LIN {X 0,Y 531.84,Z 443.101,A -85,B 0,C 180,E1 -4218.016,E2 -4218.016} C_VEL
LIN {X 0,Y 531.604,Z 454.409,A -85,B 0,C 180,E1 -4218.756,E2 -4218.756} C_VEL
LIN {X 0,Y 531.318,Z 464.837,A -85,B 0,C 180,E1 -4219.618,E2 -4219.618} C_VEL
LIN {X 0,Y 531.073,Z 475.093,A -85,B 0,C 180,E1 -4220.671,E2 -4220.671} C_VEL
LIN {X 0,Y 530.873,Z 483.99,A -85,B 0,C 180,E1 -4221.819,E2 -4221.819} C_VEL
LIN {X 0,Y 530.696,Z 491.14,A -85,B 0,C 180,E1 -4222.965,E2 -4222.965} C_VEL
LIN {X 0,Y 530.656,Z 495.995,A -85,B 0,C 180,E1 -4223.919,E2 -4223.919} C_VEL
LIN {X 0,Y 530.466,Z 500.698,A -85,B 0,C 180,E1 -4225.061,E2 -4225.061} C_VEL
LIN {X 0,Y 530.516,Z 504.289,A -85,B 0,C 180,E1 -4226.203,E2 -4226.203} C_VEL
LIN {X 0,Y 530.512,Z 506.139,A -85,B 0,C 180,E1 -4226.963,E2 -4226.963} C_VEL
LIN {X 0,Y 530.412,Z 507.563,A -85,B 0,C 180,E1 -4227.723,E2 -4227.723} C_VEL
LIN {X 0,Y 530.351,Z 509.173,A -85,B 0,C 180,E1 -4229.241,E2 -4229.241} C_VEL
LIN {X 0,Y 530.351,Z 509.411,A -85,B 0,C 180,E1 -4230.001,E2 -4230.001} C_VEL
LIN {X 0,Y 530.35,Z 509.227,A -85,B 0,C 180,E1 -4230.76,E2 -4230.76} C_VEL
LIN {X 0,Y 530.413,Z 507.691,A -85,B 0,C 180,E1 -4232.279,E2 -4232.279} C_VEL
LIN {X 0,Y 530.513,Z 506.338,A -85,B 0,C 180,E1 -4233.038,E2 -4233.038} C_VEL
LIN {X 0,Y 530.524,Z 503.495,A -85,B 0,C 180,E1 -4234.179,E2 -4234.179} C_VEL
LIN {X 0,Y 530.524,Z 499.631,A -85,B 0,C 180,E1 -4235.321,E2 -4235.321} C_VEL
LIN {X 0,Y 530.634,Z 493.865,A -85,B 0,C 180,E1 -4236.614,E2 -4236.614} C_VEL
LIN {X 0,Y 530.793,Z 487.123,A -85,B 0,C 180,E1 -4237.801,E2 -4237.801} C_VEL
LIN {X 0,Y 530.99,Z 478.999,A -85,B 0,C 180,E1 -4238.948,E2 -4238.948} C_VEL
LIN {X 0,Y 531.181,Z 470.63,A -85,B 0,C 180,E1 -4239.905,E2 -4239.905} C_VEL
LIN {X 0,Y 531.448,Z 460.37,A -85,B 0,C 180,E1 -4240.863,E2 -4240.863} C_VEL
LIN {X 0,Y 531.706,Z 449.647,A -85,B 0,C 180,E1 -4241.669,E2 -4241.669} C_VEL
LIN {X 0,Y 531.929,Z 439.01,A -85,B 0,C 180,E1 -4242.302,E2 -4242.302} C_VEL
LIN {X 0,Y 532.142,Z 426.406,A -85,B 0,C 180,E1 -4242.878,E2 -4242.878} C_VEL
LIN {X 0,Y 532.35,Z 413.949,A -85,B 0,C 180,E1 -4243.286,E2 -4243.286} C_VEL
LIN {X 0,Y 532.493,Z 401.048,A -85,B 0,C 180,E1 -4243.549,E2 -4243.549} C_VEL
LIN {X 0,Y 532.729,Z 307.619,A -85,B 0,C 180,E1 -4244.818,E2 -4244.818} C_VEL
LIN {X 0,Y 530.943,Z 296.994,A -85,B 0,C 180,E1 -4245.036,E2 -4245.036} C_VEL
LIN {X 0,Y 530.99,Z 279.347,A -85,B 0,C 180,E1 -4247.614,E2 -4247.614} C_VEL
LIN {X 0,Y 531.03,Z 279.335,A -85,B 0,C 180,E1 -4250.128,E2 -4250.128} C_VEL
LIN {X 0,Y 530.951,Z 279.344,A -85,B 0,C 180,E1 -4252.574,E2 -4252.574} C_VEL
LIN {X 0,Y 530.994,Z 279.343,A -85,B 0,C 180,E1 -4255.059,E2 -4255.059} C_VEL
LIN {X 0,Y 531.014,Z 279.341,A -85,B 0,C 180,E1 -4257.596,E2 -4257.596} C_VEL
LIN {X 0,Y 530.971,Z 279.342,A -85,B 0,C 180,E1 -4260.644,E2 -4260.644} C_VEL
LIN {X 0,Y 530.967,Z 279.347,A -85,B 0,C 180,E1 -4263.5,E2 -4263.5} C_VEL
LIN {X 0,Y 530.96,Z 279.344,A -85,B 0,C 180,E1 -4266.559,E2 -4266.559} C_VEL
LIN {X 0,Y 530.99,Z 279.343,A -85,B 0,C 180,E1 -4269.444,E2 -4269.444} C_VEL
LIN {X 0,Y 530.983,Z 279.341,A -85,B 0,C 180,E1 -4272.457,E2 -4272.457} C_VEL
LIN {X 0,Y 530.988,Z 279.34,A -85,B 0,C 180,E1 -4275.622,E2 -4275.622} C_VEL
LIN {X 0,Y 530.998,Z 279.341,A -85,B 0,C 180,E1 -4278.565,E2 -4278.565} C_VEL
LIN {X 0,Y 530.963,Z 279.343,A -85,B 0,C 180,E1 -4281.53,E2 -4281.53} C_VEL
LIN {X 0,Y 530.959,Z 279.344,A -85,B 0,C 180,E1 -4284.38,E2 -4284.38} C_VEL
LIN {X 0,Y 530.972,Z 279.345,A -85,B 0,C 180,E1 -4287.134,E2 -4287.134} C_VEL
LIN {X 0,Y 530.973,Z 279.34,A -85,B 0,C 180,E1 -4289.803,E2 -4289.803} C_VEL
LIN {X 0,Y 531.013,Z 279.34,A -85,B 0,C 180,E1 -4292.469,E2 -4292.469} C_VEL
LIN {X 0,Y 530.994,Z 279.343,A -85,B 0,C 180,E1 -4294.942,E2 -4294.942} C_VEL
LIN {X 0,Y 530.976,Z 279.343,A -85,B 0,C 180,E1 -4298.247,E2 -4298.247} C_VEL
LIN {X 0,Y 531.029,Z 279.405,A -85,B 0,C 180,E1 -4301.03,E2 -4301.03} C_VEL
LIN {X 0,Y 531.428,Z 285.13,A -85,B 0,C 180,E1 -4302.211,E2 -4302.211} C_VEL
LIN {X 0,Y 531.168,Z 299.568,A -85,B 0,C 180,E1 -4305.116,E2 -4305.116} C_VEL
LIN {X 0,Y 532.806,Z 309.363,A -85,B 0,C 180,E1 -4305.312,E2 -4305.312} C_VEL
LIN {X 0,Y 532.304,Z 405.637,A -85,B 0,C 180,E1 -4306.665,E2 -4306.665} C_VEL
LIN {X 0,Y 532.214,Z 419.063,A -85,B 0,C 180,E1 -4307.003,E2 -4307.003} C_VEL
LIN {X 0,Y 531.973,Z 431.141,A -85,B 0,C 180,E1 -4307.458,E2 -4307.458} C_VEL
LIN {X 0,Y 531.773,Z 443.346,A -85,B 0,C 180,E1 -4308.079,E2 -4308.079} C_VEL
LIN {X 0,Y 531.504,Z 456.293,A -85,B 0,C 180,E1 -4308.946,E2 -4308.946} C_VEL
LIN {X 0,Y 531.274,Z 465.371,A -85,B 0,C 180,E1 -4309.713,E2 -4309.713} C_VEL
LIN {X 0,Y 531.065,Z 474.673,A -85,B 0,C 180,E1 -4310.67,E2 -4310.67} C_VEL
LIN {X 0,Y 530.876,Z 482.343,A -85,B 0,C 180,E1 -4311.627,E2 -4311.627} C_VEL
LIN {X 0,Y 530.723,Z 489.883,A -85,B 0,C 180,E1 -4312.773,E2 -4312.773} C_VEL
LIN {X 0,Y 530.644,Z 495.898,A -85,B 0,C 180,E1 -4313.918,E2 -4313.918} C_VEL
LIN {X 0,Y 530.473,Z 500.651,A -85,B 0,C 180,E1 -4315.06,E2 -4315.06} C_VEL
LIN {X 0,Y 530.517,Z 504.276,A -85,B 0,C 180,E1 -4316.202,E2 -4316.202} C_VEL
LIN {X 0,Y 530.512,Z 506.099,A -85,B 0,C 180,E1 -4316.962,E2 -4316.962} C_VEL
LIN {X 0,Y 530.362,Z 508.579,A -85,B 0,C 180,E1 -4318.481,E2 -4318.481} C_VEL
LIN {X 0,Y 530.352,Z 509.18,A -85,B 0,C 180,E1 -4319.241,E2 -4319.241} C_VEL
LIN {X 0,Y 530.352,Z 509.246,A -85,B 0,C 180,E1 -4320.759,E2 -4320.759} C_VEL
LIN {X 0,Y 530.362,Z 508.673,A -85,B 0,C 180,E1 -4321.519,E2 -4321.519} C_VEL
LIN {X 0,Y 530.513,Z 506.338,A -85,B 0,C 180,E1 -4323.038,E2 -4323.038} C_VEL
LIN {X 0,Y 530.524,Z 503.472,A -85,B 0,C 180,E1 -4324.178,E2 -4324.178} C_VEL
LIN {X 0,Y 530.524,Z 499.567,A -85,B 0,C 180,E1 -4325.321,E2 -4325.321} C_VEL
LIN {X 0,Y 530.618,Z 495.221,A -85,B 0,C 180,E1 -4326.325,E2 -4326.325} C_VEL
LIN {X 0,Y 530.73,Z 489.328,A -85,B 0,C 180,E1 -4327.418,E2 -4327.418} C_VEL
LIN {X 0,Y 530.853,Z 483.075,A -85,B 0,C 180,E1 -4328.374,E2 -4328.374} C_VEL
LIN {X 0,Y 531.05,Z 475.529,A -85,B 0,C 180,E1 -4329.33,E2 -4329.33} C_VEL
LIN {X 0,Y 531.24,Z 466.368,A -85,B 0,C 180,E1 -4330.288,E2 -4330.288} C_VEL
LIN {X 0,Y 531.521,Z 456.247,A -85,B 0,C 180,E1 -4331.15,E2 -4331.15} C_VEL
LIN {X 0,Y 531.755,Z 444.083,A -85,B 0,C 180,E1 -4331.968,E2 -4331.968} C_VEL
LIN {X 0,Y 531.941,Z 431.979,A -85,B 0,C 180,E1 -4332.591,E2 -4332.591} C_VEL
LIN {X 0,Y 532.15,Z 418.568,A -85,B 0,C 180,E1 -4333.096,E2 -4333.096} C_VEL
LIN {X 0,Y 532.315,Z 406.003,A -85,B 0,C 180,E1 -4333.407,E2 -4333.407} C_VEL
LIN {X 0,Y 532.63,Z 307.356,A -85,B 0,C 180,E1 -4334.813,E2 -4334.813} C_VEL
LIN {X 0,Y 531.242,Z 300.133,A -85,B 0,C 180,E1 -4334.97,E2 -4334.97} C_VEL
LIN {X 0,Y 531.56,Z 285.055,A -85,B 0,C 180,E1 -4338.062,E2 -4338.062} C_VEL
LIN {X 0,Y 531.04,Z 279.34,A -85,B 0,C 180,E1 -4339.321,E2 -4339.321} C_VEL
LIN {X 0,Y 530.98,Z 279.343,A -85,B 0,C 180,E1 -4342.101,E2 -4342.101} C_VEL
LIN {X 0,Y 530.942,Z 279.352,A -85,B 0,C 180,E1 -4345.061,E2 -4345.061} C_VEL
LIN {X 0,Y 530.953,Z 279.348,A -85,B 0,C 180,E1 -4347.599,E2 -4347.599} C_VEL
LIN {X 0,Y 530.944,Z 279.349,A -85,B 0,C 180,E1 -4350.639,E2 -4350.639} C_VEL
LIN {X 0,Y 530.948,Z 279.347,A -85,B 0,C 180,E1 -4353.496,E2 -4353.496} C_VEL
LIN {X 0,Y 530.9,Z 279.351,A -85,B 0,C 180,E1 -4356.146,E2 -4356.146} C_VEL
LIN {X 0,Y 530.954,Z 279.344,A -85,B 0,C 180,E1 -4359.446,E2 -4359.446} C_VEL
LIN {X 0,Y 530.916,Z 279.354,A -85,B 0,C 180,E1 -4362.463,E2 -4362.463} C_VEL
LIN {X 0,Y 530.963,Z 279.342,A -85,B 0,C 180,E1 -4365.45,E2 -4365.45} C_VEL
LIN {X 0,Y 530.953,Z 279.35,A -85,B 0,C 180,E1 -4368.56,E2 -4368.56} C_VEL
LIN {X 0,Y 530.953,Z 279.344,A -85,B 0,C 180,E1 -4371.528,E2 -4371.528} C_VEL
LIN {X 0,Y 530.951,Z 279.351,A -85,B 0,C 180,E1 -4374.379,E2 -4374.379} C_VEL
LIN {X 0,Y 530.971,Z 279.343,A -85,B 0,C 180,E1 -4377.133,E2 -4377.133} C_VEL
LIN {X 0,Y 530.958,Z 279.352,A -85,B 0,C 180,E1 -4379.802,E2 -4379.802} C_VEL
LIN {X 0,Y 530.971,Z 279.346,A -85,B 0,C 180,E1 -4382.477,E2 -4382.477} C_VEL
LIN {X 0,Y 531.061,Z 279.462,A -85,B 0,C 180,E1 -4385.232,E2 -4385.232} C_VEL
LIN {X 0,Y 532.337,Z 287.063,A -85,B 0,C 180,E1 -4386.461,E2 -4386.461} C_VEL
LIN {X 0,Y 532.028,Z 303.307,A -85,B 0,C 180,E1 -4388.901,E2 -4388.901} C_VEL
LIN {X 0,Y 531.681,Z 322.238,A -85,B 0,C 180,E1 -4391.695,E2 -4391.695} C_VEL
LIN {X 0,Y 531.362,Z 341.292,A -85,B 0,C 180,E1 -4394.464,E2 -4394.464} C_VEL
LIN {X 0,Y 531.274,Z 345.358,A -85,B 0,C 180,E1 -4395.052,E2 -4395.052} C_VEL
LIN {X 0,Y 532.724,Z 356.776,A -85,B 0,C 180,E1 -4395.271,E2 -4395.271} C_VEL
LIN {X 0,Y 532.333,Z 452.199,A -85,B 0,C 180,E1 -4396.592,E2 -4396.592} C_VEL
LIN {X 0,Y 532.128,Z 464.759,A -85,B 0,C 180,E1 -4396.879,E2 -4396.879} C_VEL
LIN {X 0,Y 531.919,Z 478.246,A -85,B 0,C 180,E1 -4397.359,E2 -4397.359} C_VEL
LIN {X 0,Y 531.758,Z 489.353,A -85,B 0,C 180,E1 -4397.896,E2 -4397.896} C_VEL
LIN {X 0,Y 531.519,Z 500.184,A -85,B 0,C 180,E1 -4398.56,E2 -4398.56} C_VEL
LIN {X 0,Y 531.267,Z 511.362,A -85,B 0,C 180,E1 -4399.423,E2 -4399.423} C_VEL
LIN {X 0,Y 531.049,Z 520.423,A -85,B 0,C 180,E1 -4400.285,E2 -4400.285} C_VEL
LIN {X 0,Y 530.835,Z 530.246,A -85,B 0,C 180,E1 -4401.434,E2 -4401.434} C_VEL
LIN {X 0,Y 530.675,Z 538.064,A -85,B 0,C 180,E1 -4402.58,E2 -4402.58} C_VEL
LIN {X 0,Y 530.585,Z 545.242,A -85,B 0,C 180,E1 -4403.916,E2 -4403.916} C_VEL
LIN {X 0,Y 530.459,Z 550.013,A -85,B 0,C 180,E1 -4405.059,E2 -4405.059} C_VEL
LIN {X 0,Y 530.516,Z 553.668,A -85,B 0,C 180,E1 -4406.201,E2 -4406.201} C_VEL
LIN {X 0,Y 530.457,Z 555.549,A -85,B 0,C 180,E1 -4406.961,E2 -4406.961} C_VEL
LIN {X 0,Y 530.411,Z 556.955,A -85,B 0,C 180,E1 -4407.721,E2 -4407.721} C_VEL
LIN {X 0,Y 530.345,Z 558.568,A -85,B 0,C 180,E1 -4409.24,E2 -4409.24} C_VEL
LIN {X 0,Y 530.346,Z 558.788,A -85,B 0,C 180,E1 -4409.999,E2 -4409.999} C_VEL
LIN {X 0,Y 530.361,Z 557.962,A -85,B 0,C 180,E1 -4411.518,E2 -4411.518} C_VEL
LIN {X 0,Y 530.411,Z 556.964,A -85,B 0,C 180,E1 -4412.277,E2 -4412.277} C_VEL
LIN {X 0,Y 530.457,Z 555.561,A -85,B 0,C 180,E1 -4413.037,E2 -4413.037} C_VEL
LIN {X 0,Y 530.522,Z 552.614,A -85,B 0,C 180,E1 -4414.177,E2 -4414.177} C_VEL
LIN {X 0,Y 530.524,Z 548.615,A -85,B 0,C 180,E1 -4415.32,E2 -4415.32} C_VEL
LIN {X 0,Y 530.598,Z 542.845,A -85,B 0,C 180,E1 -4416.581,E2 -4416.581} C_VEL
LIN {X 0,Y 530.719,Z 535.717,A -85,B 0,C 180,E1 -4417.8,E2 -4417.8} C_VEL
LIN {X 0,Y 530.912,Z 527.353,A -85,B 0,C 180,E1 -4418.947,E2 -4418.947} C_VEL
LIN {X 0,Y 531.081,Z 518.752,A -85,B 0,C 180,E1 -4419.905,E2 -4419.905} C_VEL
LIN {X 0,Y 531.356,Z 508.129,A -85,B 0,C 180,E1 -4420.863,E2 -4420.863} C_VEL
LIN {X 0,Y 531.567,Z 497.005,A -85,B 0,C 180,E1 -4421.671,E2 -4421.671} C_VEL
LIN {X 0,Y 531.822,Z 486.007,A -85,B 0,C 180,E1 -4422.303,E2 -4422.303} C_VEL
LIN {X 0,Y 532.037,Z 473.98,A -85,B 0,C 180,E1 -4422.831,E2 -4422.831} C_VEL
LIN {X 0,Y 532.209,Z 460.97,A -85,B 0,C 180,E1 -4423.239,E2 -4423.239} C_VEL
LIN {X 0,Y 532.392,Z 447.236,A -85,B 0,C 180,E1 -4423.502,E2 -4423.502} C_VEL
LIN {X 0,Y 532.666,Z 354.778,A -85,B 0,C 180,E1 -4424.767,E2 -4424.767} C_VEL
LIN {X 0,Y 531.319,Z 345.814,A -85,B 0,C 180,E1 -4424.952,E2 -4424.952} C_VEL
LIN {X 0,Y 531.679,Z 327.116,A -85,B 0,C 180,E1 -4427.699,E2 -4427.699} C_VEL
LIN {X 0,Y 532.152,Z 305.555,A -85,B 0,C 180,E1 -4430.889,E2 -4430.889} C_VEL
LIN {X 0,Y 532.585,Z 288.083,A -85,B 0,C 180,E1 -4433.526,E2 -4433.526} C_VEL
LIN {X 0,Y 531.04,Z 279.338,A -85,B 0,C 180,E1 -4434.976,E2 -4434.976} C_VEL
LIN {X 0,Y 531.007,Z 279.341,A -85,B 0,C 180,E1 -4437.595,E2 -4437.595} C_VEL
LIN {X 0,Y 530.972,Z 279.341,A -85,B 0,C 180,E1 -4440.644,E2 -4440.644} C_VEL
LIN {X 0,Y 530.984,Z 279.345,A -85,B 0,C 180,E1 -4443.772,E2 -4443.772} C_VEL
LIN {X 0,Y 530.946,Z 279.344,A -85,B 0,C 180,E1 -4446.558,E2 -4446.558} C_VEL
LIN {X 0,Y 530.981,Z 279.343,A -85,B 0,C 180,E1 -4449.443,E2 -4449.443} C_VEL
LIN {X 0,Y 530.958,Z 279.343,A -85,B 0,C 180,E1 -4452.457,E2 -4452.457} C_VEL
LIN {X 0,Y 530.962,Z 279.347,A -85,B 0,C 180,E1 -4455.45,E2 -4455.45} C_VEL
LIN {X 0,Y 530.974,Z 279.34,A -85,B 0,C 180,E1 -4458.562,E2 -4458.562} C_VEL
LIN {X 0,Y 530.947,Z 279.352,A -85,B 0,C 180,E1 -4461.528,E2 -4461.528} C_VEL
LIN {X 0,Y 530.946,Z 279.344,A -85,B 0,C 180,E1 -4464.379,E2 -4464.379} C_VEL
LIN {X 0,Y 530.958,Z 279.348,A -85,B 0,C 180,E1 -4467.133,E2 -4467.133} C_VEL
LIN {X 0,Y 530.942,Z 279.347,A -85,B 0,C 180,E1 -4469.801,E2 -4469.801} C_VEL
LIN {X 0,Y 530.955,Z 279.344,A -85,B 0,C 180,E1 -4472.477,E2 -4472.477} C_VEL
LIN {X 0,Y 530.938,Z 279.35,A -85,B 0,C 180,E1 -4474.939,E2 -4474.939} C_VEL
LIN {X 0,Y 530.967,Z 279.342,A -85,B 0,C 180,E1 -4477.898,E2 -4477.898} C_VEL
LIN {X 0,Y 530.972,Z 279.345,A -85,B 0,C 180,E1 -4480.676,E2 -4480.676} C_VEL
LIN {X 0,Y 530.949,Z 279.351,A -85,B 0,C 180,E1 -4483.07,E2 -4483.07} C_VEL
LIN {X 0,Y 530.988,Z 279.341,A -85,B 0,C 180,E1 -4485.435,E2 -4485.435} C_VEL
LIN {X 0,Y 531.02,Z 279.34,A -85,B 0,C 180,E1 -4488.549,E2 -4488.549} C_VEL
LIN {X 0,Y 531.018,Z 279.336,A -85,B 0,C 180,E1 -4491.629,E2 -4491.629} C_VEL
LIN {X 0,Y 531.072,Z 279.335,A -85,B 0,C 180,E1 -4494.685,E2 -4494.685} C_VEL
LIN {X 0,Y 531.113,Z 279.324,A -85,B 0,C 180,E1 -4497.725,E2 -4497.725} C_VEL
LIN {X 0,Y 531.138,Z 279.325,A -85,B 0,C 180,E1 -4500.758,E2 -4500.758} C_VEL
LIN {X 0,Y 531.045,Z 279.334,A -85,B 0,C 180,E1 -4503.035,E2 -4503.035} C_VEL
LIN {X 0,Y 531.031,Z 279.339,A -85,B 0,C 180,E1 -4506.078,E2 -4506.078} C_VEL
LIN {X 0,Y 530.996,Z 279.339,A -85,B 0,C 180,E1 -4509.139,E2 -4509.139} C_VEL
LIN {X 0,Y 531.039,Z 279.336,A -85,B 0,C 180,E1 -4511.67,E2 -4511.67} C_VEL
LIN {X 0,Y 531.014,Z 279.337,A -85,B 0,C 180,E1 -4514.953,E2 -4514.953} C_VEL
LIN {X 0,Y 530.971,Z 279.347,A -85,B 0,C 180,E1 -4517.724,E2 -4517.724} C_VEL
LIN {X 0,Y 531.016,Z 279.342,A -85,B 0,C 180,E1 -4520.128,E2 -4520.128} C_VEL
LIN {X 0,Y 530.936,Z 279.347,A -85,B 0,C 180,E1 -4522.574,E2 -4522.574} C_VEL
LIN {X 0,Y 530.978,Z 279.342,A -85,B 0,C 180,E1 -4525.059,E2 -4525.059} C_VEL
LIN {X 0,Y 530.957,Z 279.349,A -85,B 0,C 180,E1 -4527.599,E2 -4527.599} C_VEL
LIN {X 0,Y 530.953,Z 279.346,A -85,B 0,C 180,E1 -4530.198,E2 -4530.198} C_VEL
LIN {X 0,Y 530.96,Z 279.344,A -85,B 0,C 180,E1 -4532.867,E2 -4532.867} C_VEL
LIN {X 0,Y 530.943,Z 279.351,A -85,B 0,C 180,E1 -4535.621,E2 -4535.621} C_VEL
LIN {X 0,Y 530.957,Z 279.344,A -85,B 0,C 180,E1 -4538.654,E2 -4538.654} C_VEL
LIN {X 0,Y 530.983,Z 279.346,A -85,B 0,C 180,E1 -4541.437,E2 -4541.437} C_VEL
LIN {X 0,Y 530.937,Z 279.35,A -85,B 0,C 180,E1 -4543.56,E2 -4543.56} C_VEL
LIN {X 0,Y 530.27,Z 279.43,A -85,B 0,C 180,E1 -4544.193,E2 -4544.193} C_VEL
LIN {X 0,Y 527.427,Z 279.789,A -85,B 0,C 180,E1 -4545.222,E2 -4545.222} C_VEL
LIN {X 0,Y 525.026,Z 280.088,A -85,B 0,C 180,E1 -4546.051,E2 -4546.051} C_VEL
LIN {X 0,Y 523.995,Z 280.215,A -85,B 0,C 180,E1 -4546.691,E2 -4546.691} C_VEL
LIN {X 0,Y 523.91,Z 280.225,A -85,B 0,C 180,E1 -4546.907,E2 -4546.907} C_VEL
LIN {X 0,Y 523.945,Z 280.218,A -85,B 0,C 180,E1 -4549.922,E2 -4549.922} C_VEL
LIN {X 0,Y 523.904,Z 280.228,A -85,B 0,C 180,E1 -4552.869,E2 -4552.869} C_VEL
LIN {X 0,Y 523.917,Z 280.222,A -85,B 0,C 180,E1 -4555.71,E2 -4555.71} C_VEL
LIN {X 0,Y 523.917,Z 280.223,A -85,B 0,C 180,E1 -4558.457,E2 -4558.457} C_VEL
LIN {X 0,Y 523.928,Z 280.224,A -85,B 0,C 180,E1 -4561.126,E2 -4561.126} C_VEL
LIN {X 0,Y 523.983,Z 280.213,A -85,B 0,C 180,E1 -4563.981,E2 -4563.981} C_VEL
LIN {X 0,Y 523.911,Z 280.225,A -85,B 0,C 180,E1 -4567.107,E2 -4567.107} C_VEL
LIN {X 0,Y 523.979,Z 280.213,A -85,B 0,C 180,E1 -4569.867,E2 -4569.867} C_VEL
LIN {X 0,Y 523.902,Z 280.231,A -85,B 0,C 180,E1 -4572.601,E2 -4572.601} C_VEL
LIN {X 0,Y 523.873,Z 295.889,A -85,B 0,C 180,E1 -4574.771,E2 -4574.771} C_VEL
LIN {X 0,Y 523.904,Z 296.55,A -85,B 0,C 180,E1 -4574.856,E2 -4574.856} C_VEL
LIN {X 0,Y 525.989,Z 309.337,A -85,B 0,C 180,E1 -4575.099,E2 -4575.099} C_VEL
LIN {X 0,Y 525.543,Z 405.952,A -85,B 0,C 180,E1 -4576.442,E2 -4576.442} C_VEL
LIN {X 0,Y 525.379,Z 419.475,A -85,B 0,C 180,E1 -4576.782,E2 -4576.782} C_VEL
LIN {X 0,Y 525.135,Z 431.546,A -85,B 0,C 180,E1 -4577.243,E2 -4577.243} C_VEL
LIN {X 0,Y 524.898,Z 444.027,A -85,B 0,C 180,E1 -4577.892,E2 -4577.892} C_VEL
LIN {X 0,Y 524.661,Z 454.714,A -85,B 0,C 180,E1 -4578.605,E2 -4578.605} C_VEL
LIN {X 0,Y 524.33,Z 465.146,A -85,B 0,C 180,E1 -4579.478,E2 -4579.478} C_VEL
LIN {X 0,Y 524.078,Z 475.405,A -85,B 0,C 180,E1 -4580.546,E2 -4580.546} C_VEL
LIN {X 0,Y 523.84,Z 484.305,A -85,B 0,C 180,E1 -4581.708,E2 -4581.708} C_VEL
LIN {X 0,Y 523.659,Z 491.456,A -85,B 0,C 180,E1 -4582.87,E2 -4582.87} C_VEL
LIN {X 0,Y 523.601,Z 496.312,A -85,B 0,C 180,E1 -4583.837,E2 -4583.837} C_VEL
LIN {X 0,Y 523.392,Z 501.016,A -85,B 0,C 180,E1 -4584.994,E2 -4584.994} C_VEL
LIN {X 0,Y 523.443,Z 504.606,A -85,B 0,C 180,E1 -4586.152,E2 -4586.152} C_VEL
LIN {X 0,Y 523.446,Z 506.456,A -85,B 0,C 180,E1 -4586.922,E2 -4586.922} C_VEL
LIN {X 0,Y 523.338,Z 507.88,A -85,B 0,C 180,E1 -4587.692,E2 -4587.692} C_VEL
LIN {X 0,Y 523.259,Z 509.49,A -85,B 0,C 180,E1 -4589.231,E2 -4589.231} C_VEL
LIN {X 0,Y 523.259,Z 509.728,A -85,B 0,C 180,E1 -4590.001,E2 -4590.001} C_VEL
LIN {X 0,Y 523.258,Z 509.544,A -85,B 0,C 180,E1 -4590.77,E2 -4590.77} C_VEL
LIN {X 0,Y 523.338,Z 508.006,A -85,B 0,C 180,E1 -4592.31,E2 -4592.31} C_VEL
LIN {X 0,Y 523.447,Z 506.652,A -85,B 0,C 180,E1 -4593.079,E2 -4593.079} C_VEL
LIN {X 0,Y 523.449,Z 503.809,A -85,B 0,C 180,E1 -4594.236,E2 -4594.236} C_VEL
LIN {X 0,Y 523.464,Z 499.943,A -85,B 0,C 180,E1 -4595.393,E2 -4595.393} C_VEL
LIN {X 0,Y 523.564,Z 494.602,A -85,B 0,C 180,E1 -4596.619,E2 -4596.619} C_VEL
LIN {X 0,Y 523.773,Z 487.431,A -85,B 0,C 180,E1 -4597.906,E2 -4597.906} C_VEL
LIN {X 0,Y 523.965,Z 479.304,A -85,B 0,C 180,E1 -4599.069,E2 -4599.069} C_VEL
LIN {X 0,Y 524.188,Z 470.929,A -85,B 0,C 180,E1 -4600.038,E2 -4600.038} C_VEL
LIN {X 0,Y 524.483,Z 460.663,A -85,B 0,C 180,E1 -4601.009,E2 -4601.009} C_VEL
LIN {X 0,Y 524.751,Z 450.206,A -85,B 0,C 180,E1 -4601.807,E2 -4601.807} C_VEL
LIN {X 0,Y 525.008,Z 439.281,A -85,B 0,C 180,E1 -4602.466,E2 -4602.466} C_VEL
LIN {X 0,Y 525.243,Z 426.658,A -85,B 0,C 180,E1 -4603.05,E2 -4603.05} C_VEL
LIN {X 0,Y 525.47,Z 414.157,A -85,B 0,C 180,E1 -4603.463,E2 -4603.463} C_VEL
LIN {X 0,Y 525.606,Z 401.164,A -85,B 0,C 180,E1 -4603.73,E2 -4603.73} C_VEL
LIN {X 0,Y 525.987,Z 309.161,A -85,B 0,C 180,E1 -4604.993,E2 -4604.993} C_VEL
LIN {X 0,Y 523.876,Z 296.59,A -85,B 0,C 180,E1 -4605.233,E2 -4605.233} C_VEL
LIN {X 0,Y 523.869,Z 281.402,A -85,B 0,C 180,E1 -4607.318,E2 -4607.318} C_VEL
LIN {X 0,Y 523.867,Z 280.235,A -85,B 0,C 180,E1 -4607.514,E2 -4607.514} C_VEL
LIN {X 0,Y 523.984,Z 280.213,A -85,B 0,C 180,E1 -4610.134,E2 -4610.134} C_VEL
LIN {X 0,Y 523.916,Z 280.223,A -85,B 0,C 180,E1 -4612.894,E2 -4612.894} C_VEL
LIN {X 0,Y 523.988,Z 280.212,A -85,B 0,C 180,E1 -4616.02,E2 -4616.02} C_VEL
LIN {X 0,Y 523.934,Z 280.221,A -85,B 0,C 180,E1 -4618.876,E2 -4618.876} C_VEL
LIN {X 0,Y 523.924,Z 280.224,A -85,B 0,C 180,E1 -4621.545,E2 -4621.545} C_VEL
LIN {X 0,Y 523.925,Z 280.219,A -85,B 0,C 180,E1 -4624.292,E2 -4624.292} C_VEL
LIN {X 0,Y 523.912,Z 280.227,A -85,B 0,C 180,E1 -4627.133,E2 -4627.133} C_VEL
LIN {X 0,Y 523.943,Z 280.217,A -85,B 0,C 180,E1 -4630.13,E2 -4630.13} C_VEL
LIN {X 0,Y 523.927,Z 280.226,A -85,B 0,C 180,E1 -4633.167,E2 -4633.167} C_VEL
LIN {X 0,Y 523.941,Z 280.217,A -85,B 0,C 180,E1 -4635.772,E2 -4635.772} C_VEL
LIN {X 0,Y 523.944,Z 280.223,A -85,B 0,C 180,E1 -4638.908,E2 -4638.908} C_VEL
LIN {X 0,Y 523.921,Z 280.219,A -85,B 0,C 180,E1 -4641.898,E2 -4641.898} C_VEL
LIN {X 0,Y 523.929,Z 280.226,A -85,B 0,C 180,E1 -4644.911,E2 -4644.911} C_VEL
LIN {X 0,Y 523.94,Z 280.216,A -85,B 0,C 180,E1 -4647.68,E2 -4647.68} C_VEL
LIN {X 0,Y 523.958,Z 280.221,A -85,B 0,C 180,E1 -4650.677,E2 -4650.677} C_VEL
LIN {X 0,Y 523.95,Z 280.222,A -85,B 0,C 180,E1 -4652.867,E2 -4652.867} C_VEL
LIN {X 0,Y 523.946,Z 280.215,A -85,B 0,C 180,E1 -4655.802,E2 -4655.802} C_VEL
LIN {X 0,Y 523.95,Z 280.223,A -85,B 0,C 180,E1 -4658.767,E2 -4658.767} C_VEL
LIN {X 0,Y 523.994,Z 280.322,A -85,B 0,C 180,E1 -4660.918,E2 -4660.918} C_VEL
LIN {X 0,Y 524.447,Z 285.856,A -85,B 0,C 180,E1 -4662.075,E2 -4662.075} C_VEL
LIN {X 0,Y 524.182,Z 299.819,A -85,B 0,C 180,E1 -4664.913,E2 -4664.913} C_VEL
LIN {X 0,Y 525.952,Z 309.464,A -85,B 0,C 180,E1 -4665.116,E2 -4665.116} C_VEL
LIN {X 0,Y 525.383,Z 406.411,A -85,B 0,C 180,E1 -4666.511,E2 -4666.511} C_VEL
LIN {X 0,Y 525.278,Z 420.296,A -85,B 0,C 180,E1 -4666.877,E2 -4666.877} C_VEL
LIN {X 0,Y 525.013,Z 432.131,A -85,B 0,C 180,E1 -4667.338,E2 -4667.338} C_VEL
LIN {X 0,Y 524.795,Z 444.278,A -85,B 0,C 180,E1 -4667.974,E2 -4667.974} C_VEL
LIN {X 0,Y 524.536,Z 456.361,A -85,B 0,C 180,E1 -4668.797,E2 -4668.797} C_VEL
LIN {X 0,Y 524.265,Z 465.51,A -85,B 0,C 180,E1 -4669.573,E2 -4669.573} C_VEL
LIN {X 0,Y 524.036,Z 474.853,A -85,B 0,C 180,E1 -4670.544,E2 -4670.544} C_VEL
LIN {X 0,Y 523.857,Z 482.554,A -85,B 0,C 180,E1 -4671.514,E2 -4671.514} C_VEL
LIN {X 0,Y 523.665,Z 490.107,A -85,B 0,C 180,E1 -4672.675,E2 -4672.675} C_VEL
LIN {X 0,Y 523.577,Z 496.146,A -85,B 0,C 180,E1 -4673.835,E2 -4673.835} C_VEL
LIN {X 0,Y 523.395,Z 500.92,A -85,B 0,C 180,E1 -4674.993,E2 -4674.993} C_VEL
LIN {X 0,Y 523.444,Z 504.566,A -85,B 0,C 180,E1 -4676.151,E2 -4676.151} C_VEL
LIN {X 0,Y 523.447,Z 506.412,A -85,B 0,C 180,E1 -4676.921,E2 -4676.921} C_VEL
LIN {X 0,Y 523.275,Z 508.897,A -85,B 0,C 180,E1 -4678.461,E2 -4678.461} C_VEL
LIN {X 0,Y 523.261,Z 509.51,A -85,B 0,C 180,E1 -4679.23,E2 -4679.23} C_VEL
LIN {X 0,Y 523.26,Z 509.579,A -85,B 0,C 180,E1 -4680.77,E2 -4680.77} C_VEL
LIN {X 0,Y 523.275,Z 509.011,A -85,B 0,C 180,E1 -4681.539,E2 -4681.539} C_VEL
LIN {X 0,Y 523.447,Z 506.667,A -85,B 0,C 180,E1 -4683.079,E2 -4683.079} C_VEL
LIN {X 0,Y 523.449,Z 503.793,A -85,B 0,C 180,E1 -4684.235,E2 -4684.235} C_VEL
LIN {X 0,Y 523.463,Z 499.875,A -85,B 0,C 180,E1 -4685.393,E2 -4685.393} C_VEL
LIN {X 0,Y 523.561,Z 494.486,A -85,B 0,C 180,E1 -4686.615,E2 -4686.615} C_VEL
LIN {X 0,Y 523.705,Z 488.418,A -85,B 0,C 180,E1 -4687.712,E2 -4687.712} C_VEL
LIN {X 0,Y 523.924,Z 480.451,A -85,B 0,C 180,E1 -4688.874,E2 -4688.874} C_VEL
LIN {X 0,Y 524.13,Z 472.277,A -85,B 0,C 180,E1 -4689.844,E2 -4689.844} C_VEL
LIN {X 0,Y 524.369,Z 462.263,A -85,B 0,C 180,E1 -4690.815,E2 -4690.815} C_VEL
LIN {X 0,Y 524.666,Z 450.855,A -85,B 0,C 180,E1 -4691.692,E2 -4691.692} C_VEL
LIN {X 0,Y 524.896,Z 439.732,A -85,B 0,C 180,E1 -4692.37,E2 -4692.37} C_VEL
LIN {X 0,Y 525.098,Z 428.425,A -85,B 0,C 180,E1 -4692.906,E2 -4692.906} C_VEL
LIN {X 0,Y 525.291,Z 415.626,A -85,B 0,C 180,E1 -4693.344,E2 -4693.344} C_VEL
LIN {X 0,Y 525.4,Z 402.166,A -85,B 0,C 180,E1 -4693.636,E2 -4693.636} C_VEL
LIN {X 0,Y 525.898,Z 308.914,A -85,B 0,C 180,E1 -4694.982,E2 -4694.982} C_VEL
LIN {X 0,Y 524.283,Z 300.578,A -85,B 0,C 180,E1 -4695.168,E2 -4695.168} C_VEL
LIN {X 0,Y 524.6,Z 287.041,A -85,B 0,C 180,E1 -4697.976,E2 -4697.976} C_VEL
LIN {X 0,Y 524.188,Z 281.462,A -85,B 0,C 180,E1 -4699.177,E2 -4699.177} C_VEL
LIN {X 0,Y 523.984,Z 280.219,A -85,B 0,C 180,E1 -4699.49,E2 -4699.49} C_VEL
LIN {X 0,Y 523.92,Z 280.223,A -85,B 0,C 180,E1 -4702.242,E2 -4702.242} C_VEL
LIN {X 0,Y 523.9,Z 280.225,A -85,B 0,C 180,E1 -4704.573,E2 -4704.573} C_VEL
LIN {X 0,Y 523.914,Z 280.224,A -85,B 0,C 180,E1 -4707.704,E2 -4707.704} C_VEL
LIN {X 0,Y 523.9,Z 280.228,A -85,B 0,C 180,E1 -4710.845,E2 -4710.845} C_VEL
LIN {X 0,Y 523.912,Z 280.222,A -85,B 0,C 180,E1 -4713.726,E2 -4713.726} C_VEL
LIN {X 0,Y 523.858,Z 280.23,A -85,B 0,C 180,E1 -4716.394,E2 -4716.394} C_VEL
LIN {X 0,Y 523.9,Z 280.226,A -85,B 0,C 180,E1 -4719.087,E2 -4719.087} C_VEL
LIN {X 0,Y 523.894,Z 280.225,A -85,B 0,C 180,E1 -4722.125,E2 -4722.125} C_VEL
LIN {X 0,Y 523.934,Z 280.218,A -85,B 0,C 180,E1 -4725.311,E2 -4725.311} C_VEL
LIN {X 0,Y 523.915,Z 280.226,A -85,B 0,C 180,E1 -4728.695,E2 -4728.695} C_VEL
LIN {X 0,Y 523.914,Z 280.224,A -85,B 0,C 180,E1 -4731.897,E2 -4731.897} C_VEL
LIN {X 0,Y 523.922,Z 280.221,A -85,B 0,C 180,E1 -4734.912,E2 -4734.912} C_VEL
LIN {X 0,Y 523.939,Z 280.222,A -85,B 0,C 180,E1 -4737.679,E2 -4737.679} C_VEL
LIN {X 0,Y 523.956,Z 280.221,A -85,B 0,C 180,E1 -4740.677,E2 -4740.677} C_VEL
LIN {X 0,Y 523.935,Z 280.225,A -85,B 0,C 180,E1 -4743.726,E2 -4743.726} C_VEL
LIN {X 0,Y 523.997,Z 280.266,A -85,B 0,C 180,E1 -4745.034,E2 -4745.034} C_VEL
LIN {X 0,Y 525.376,Z 288.167,A -85,B 0,C 180,E1 -4746.339,E2 -4746.339} C_VEL
LIN {X 0,Y 525.196,Z 298.895,A -85,B 0,C 180,E1 -4747.994,E2 -4747.994} C_VEL
LIN {X 0,Y 524.772,Z 316.472,A -85,B 0,C 180,E1 -4750.642,E2 -4750.642} C_VEL
LIN {X 0,Y 524.448,Z 334.09,A -85,B 0,C 180,E1 -4753.254,E2 -4753.254} C_VEL
LIN {X 0,Y 524.268,Z 344.866,A -85,B 0,C 180,E1 -4754.838,E2 -4754.838} C_VEL
LIN {X 0,Y 525.862,Z 356.746,A -85,B 0,C 180,E1 -4755.08,E2 -4755.08} C_VEL
LIN {X 0,Y 525.385,Z 453.304,A -85,B 0,C 180,E1 -4756.461,E2 -4756.461} C_VEL
LIN {X 0,Y 525.165,Z 465.949,A -85,B 0,C 180,E1 -4756.775,E2 -4756.775} C_VEL
LIN {X 0,Y 524.891,Z 479.58,A -85,B 0,C 180,E1 -4757.285,E2 -4757.285} C_VEL
LIN {X 0,Y 524.68,Z 491.736,A -85,B 0,C 180,E1 -4757.912,E2 -4757.912} C_VEL
LIN {X 0,Y 524.372,Z 503.491,A -85,B 0,C 180,E1 -4758.695,E2 -4758.695} C_VEL
LIN {X 0,Y 524.153,Z 513.999,A -85,B 0,C 180,E1 -4759.571,E2 -4759.571} C_VEL
LIN {X 0,Y 523.905,Z 523.41,A -85,B 0,C 180,E1 -4760.541,E2 -4760.541} C_VEL
LIN {X 0,Y 523.704,Z 532.525,A -85,B 0,C 180,E1 -4761.705,E2 -4761.705} C_VEL
LIN {X 0,Y 523.573,Z 539.877,A -85,B 0,C 180,E1 -4762.867,E2 -4762.867} C_VEL
LIN {X 0,Y 523.48,Z 544.816,A -85,B 0,C 180,E1 -4763.834,E2 -4763.834} C_VEL
LIN {X 0,Y 523.384,Z 549.62,A -85,B 0,C 180,E1 -4764.992,E2 -4764.992} C_VEL
LIN {X 0,Y 523.443,Z 553.296,A -85,B 0,C 180,E1 -4766.15,E2 -4766.15} C_VEL
LIN {X 0,Y 523.368,Z 555.193,A -85,B 0,C 180,E1 -4766.92,E2 -4766.92} C_VEL
LIN {X 0,Y 523.335,Z 556.609,A -85,B 0,C 180,E1 -4767.69,E2 -4767.69} C_VEL
LIN {X 0,Y 523.253,Z 558.234,A -85,B 0,C 180,E1 -4769.23,E2 -4769.23} C_VEL
LIN {X 0,Y 523.254,Z 558.459,A -85,B 0,C 180,E1 -4769.999,E2 -4769.999} C_VEL
LIN {X 0,Y 523.253,Z 558.244,A -85,B 0,C 180,E1 -4770.769,E2 -4770.769} C_VEL
LIN {X 0,Y 523.335,Z 556.634,A -85,B 0,C 180,E1 -4772.308,E2 -4772.308} C_VEL
LIN {X 0,Y 523.367,Z 555.225,A -85,B 0,C 180,E1 -4773.078,E2 -4773.078} C_VEL
LIN {X 0,Y 523.424,Z 552.267,A -85,B 0,C 180,E1 -4774.234,E2 -4774.234} C_VEL
LIN {X 0,Y 523.461,Z 548.254,A -85,B 0,C 180,E1 -4775.392,E2 -4775.392} C_VEL
LIN {X 0,Y 523.516,Z 542.961,A -85,B 0,C 180,E1 -4776.574,E2 -4776.574} C_VEL
LIN {X 0,Y 523.616,Z 536.549,A -85,B 0,C 180,E1 -4777.713,E2 -4777.713} C_VEL
LIN {X 0,Y 523.815,Z 528.418,A -85,B 0,C 180,E1 -4778.875,E2 -4778.875} C_VEL
LIN {X 0,Y 523.991,Z 520.112,A -85,B 0,C 180,E1 -4779.846,E2 -4779.846} C_VEL
LIN {X 0,Y 524.26,Z 509.962,A -85,B 0,C 180,E1 -4780.816,E2 -4780.816} C_VEL
LIN {X 0,Y 524.491,Z 499.888,A -85,B 0,C 180,E1 -4781.594,E2 -4781.594} C_VEL
LIN {X 0,Y 524.805,Z 487.169,A -85,B 0,C 180,E1 -4782.372,E2 -4782.372} C_VEL
LIN {X 0,Y 525.043,Z 475.749,A -85,B 0,C 180,E1 -4782.906,E2 -4782.906} C_VEL
LIN {X 0,Y 525.239,Z 462.748,A -85,B 0,C 180,E1 -4783.344,E2 -4783.344} C_VEL
LIN {X 0,Y 525.484,Z 449.02,A -85,B 0,C 180,E1 -4783.633,E2 -4783.633} C_VEL
LIN {X 0,Y 525.789,Z 355.511,A -85,B 0,C 180,E1 -4784.949,E2 -4784.949} C_VEL
LIN {X 0,Y 524.31,Z 345.569,A -85,B 0,C 180,E1 -4785.152,E2 -4785.152} C_VEL
LIN {X 0,Y 524.711,Z 326.407,A -85,B 0,C 180,E1 -4788.014,E2 -4788.014} C_VEL
LIN {X 0,Y 525.189,Z 306.678,A -85,B 0,C 180,E1 -4790.974,E2 -4790.974} C_VEL
LIN {X 0,Y 525.668,Z 289.237,A -85,B 0,C 180,E1 -4793.645,E2 -4793.645} C_VEL
LIN {X 0,Y 524.005,Z 280.214,A -85,B 0,C 180,E1 -4795.149,E2 -4795.149} C_VEL
LIN {X 0,Y 523.955,Z 280.223,A -85,B 0,C 180,E1 -4797.999,E2 -4797.999} C_VEL
LIN {X 0,Y 523.942,Z 280.216,A -85,B 0,C 180,E1 -4800.854,E2 -4800.854} C_VEL
LIN {X 0,Y 523.956,Z 280.22,A -85,B 0,C 180,E1 -4803.733,E2 -4803.733} C_VEL
LIN {X 0,Y 523.895,Z 280.224,A -85,B 0,C 180,E1 -4806.4,E2 -4806.4} C_VEL
LIN {X 0,Y 523.915,Z 280.22,A -85,B 0,C 180,E1 -4809.084,E2 -4809.084} C_VEL
LIN {X 0,Y 523.935,Z 280.22,A -85,B 0,C 180,E1 -4812.119,E2 -4812.119} C_VEL
LIN {X 0,Y 523.932,Z 280.221,A -85,B 0,C 180,E1 -4815.31,E2 -4815.31} C_VEL
LIN {X 0,Y 523.934,Z 280.218,A -85,B 0,C 180,E1 -4818.691,E2 -4818.691} C_VEL
LIN {X 0,Y 523.907,Z 280.224,A -85,B 0,C 180,E1 -4821.897,E2 -4821.897} C_VEL
LIN {X 0,Y 523.916,Z 280.223,A -85,B 0,C 180,E1 -4824.911,E2 -4824.911} C_VEL
LIN {X 0,Y 523.927,Z 280.222,A -85,B 0,C 180,E1 -4827.679,E2 -4827.679} C_VEL
LIN {X 0,Y 523.927,Z 280.221,A -85,B 0,C 180,E1 -4830.68,E2 -4830.68} C_VEL
LIN {X 0,Y 523.892,Z 280.225,A -85,B 0,C 180,E1 -4833.724,E2 -4833.724} C_VEL
LIN {X 0,Y 523.898,Z 280.223,A -85,B 0,C 180,E1 -4836.269,E2 -4836.269} C_VEL
LIN {X 0,Y 523.933,Z 280.222,A -85,B 0,C 180,E1 -4838.766,E2 -4838.766} C_VEL
LIN {X 0,Y 523.927,Z 280.224,A -85,B 0,C 180,E1 -4841.22,E2 -4841.22} C_VEL
LIN {X 0,Y 523.898,Z 280.223,A -85,B 0,C 180,E1 -4843.638,E2 -4843.638} C_VEL
LIN {X 0,Y 523.901,Z 280.223,A -85,B 0,C 180,E1 -4846.027,E2 -4846.027} C_VEL
LIN {X 0,Y 524.004,Z 280.213,A -85,B 0,C 180,E1 -4848.394,E2 -4848.394} C_VEL
LIN {X 0,Y 523.971,Z 280.214,A -85,B 0,C 180,E1 -4851.515,E2 -4851.515} C_VEL
LIN {X 0,Y 524.018,Z 280.213,A -85,B 0,C 180,E1 -4854.613,E2 -4854.613} C_VEL
LIN {X 0,Y 524.086,Z 280.2,A -85,B 0,C 180,E1 -4857.694,E2 -4857.694} C_VEL
LIN {X 0,Y 524.108,Z 280.201,A -85,B 0,C 180,E1 -4860.768,E2 -4860.768} C_VEL
LIN {X 0,Y 523.988,Z 280.213,A -85,B 0,C 180,E1 -4863.075,E2 -4863.075} C_VEL
LIN {X 0,Y 523.993,Z 280.216,A -85,B 0,C 180,E1 -4866.16,E2 -4866.16} C_VEL
LIN {X 0,Y 523.967,Z 280.215,A -85,B 0,C 180,E1 -4869.263,E2 -4869.263} C_VEL
LIN {X 0,Y 523.989,Z 280.215,A -85,B 0,C 180,E1 -4871.737,E2 -4871.737} C_VEL
LIN {X 0,Y 523.977,Z 280.213,A -85,B 0,C 180,E1 -4875.05,E2 -4875.05} C_VEL
LIN {X 0,Y 523.935,Z 280.223,A -85,B 0,C 180,E1 -4877.97,E2 -4877.97} C_VEL
LIN {X 0,Y 523.949,Z 280.219,A -85,B 0,C 180,E1 -4880.411,E2 -4880.411} C_VEL
LIN {X 0,Y 523.901,Z 280.223,A -85,B 0,C 180,E1 -4882.894,E2 -4882.894} C_VEL
LIN {X 0,Y 523.918,Z 280.224,A -85,B 0,C 180,E1 -4885.421,E2 -4885.421} C_VEL
LIN {X 0,Y 523.907,Z 280.227,A -85,B 0,C 180,E1 -4888.003,E2 -4888.003} C_VEL
LIN {X 0,Y 523.932,Z 280.219,A -85,B 0,C 180,E1 -4890.854,E2 -4890.854} C_VEL
LIN {X 0,Y 523.952,Z 280.221,A -85,B 0,C 180,E1 -4893.735,E2 -4893.735} C_VEL
LIN {X 0,Y 523.892,Z 280.224,A -85,B 0,C 180,E1 -4896.401,E2 -4896.401} C_VEL
LIN {X 0,Y 523.913,Z 280.225,A -85,B 0,C 180,E1 -4899.086,E2 -4899.086} C_VEL
LIN {X 0,Y 523.936,Z 280.219,A -85,B 0,C 180,E1 -4902.121,E2 -4902.121} C_VEL
LIN {X 0,Y 523.938,Z 280.223,A -85,B 0,C 180,E1 -4905.311,E2 -4905.311} C_VEL
LIN {X 0,Y 523.91,Z 280.225,A -85,B 0,C 180,E1 -4906.907,E2 -4906.907} C_VEL
LIN {X 0,Y 523.246,Z 280.309,A -85,B 0,C 180,E1 -4907.549,E2 -4907.549} C_VEL
LIN {X 0,Y 520.406,Z 280.66,A -85,B 0,C 180,E1 -4908.59,E2 -4908.59} C_VEL
LIN {X 0,Y 518.002,Z 280.962,A -85,B 0,C 180,E1 -4909.429,E2 -4909.429} C_VEL
LIN {X 0,Y 516.965,Z 281.087,A -85,B 0,C 180,E1 -4910.077,E2 -4910.077} C_VEL
LIN {X 0,Y 516.877,Z 281.098,A -85,B 0,C 180,E1 -4910.296,E2 -4910.296} C_VEL
LIN {X 0,Y 516.874,Z 281.102,A -85,B 0,C 180,E1 -4913.344,E2 -4913.344} C_VEL
LIN {X 0,Y 516.881,Z 281.098,A -85,B 0,C 180,E1 -4916.12,E2 -4916.12} C_VEL
LIN {X 0,Y 516.887,Z 281.101,A -85,B 0,C 180,E1 -4918.937,E2 -4918.937} C_VEL
LIN {X 0,Y 516.909,Z 281.095,A -85,B 0,C 180,E1 -4921.585,E2 -4921.585} C_VEL
LIN {X 0,Y 516.929,Z 281.093,A -85,B 0,C 180,E1 -4924.212,E2 -4924.212} C_VEL
LIN {X 0,Y 516.86,Z 281.107,A -85,B 0,C 180,E1 -4926.777,E2 -4926.777} C_VEL
LIN {X 0,Y 516.94,Z 281.09,A -85,B 0,C 180,E1 -4929.733,E2 -4929.733} C_VEL
LIN {X 0,Y 516.863,Z 281.108,A -85,B 0,C 180,E1 -4932.595,E2 -4932.595} C_VEL
LIN {X 0,Y 516.791,Z 281.352,A -85,B 0,C 180,E1 -4932.745,E2 -4932.745} C_VEL
LIN {X 0,Y 516.778,Z 292.491,A -85,B 0,C 180,E1 -4934.218,E2 -4934.218} C_VEL
LIN {X 0,Y 516.841,Z 296.106,A -85,B 0,C 180,E1 -4934.638,E2 -4934.638} C_VEL
LIN {X 0,Y 519.151,Z 311.086,A -85,B 0,C 180,E1 -4934.92,E2 -4934.92} C_VEL
LIN {X 0,Y 518.659,Z 406.169,A -85,B 0,C 180,E1 -4936.259,E2 -4936.259} C_VEL
LIN {X 0,Y 518.475,Z 419.738,A -85,B 0,C 180,E1 -4936.603,E2 -4936.603} C_VEL
LIN {X 0,Y 518.22,Z 431.831,A -85,B 0,C 180,E1 -4937.07,E2 -4937.07} C_VEL
LIN {X 0,Y 518.016,Z 442.91,A -85,B 0,C 180,E1 -4937.644,E2 -4937.644} C_VEL
LIN {X 0,Y 517.761,Z 453.66,A -85,B 0,C 180,E1 -4938.352,E2 -4938.352} C_VEL
LIN {X 0,Y 517.41,Z 464.425,A -85,B 0,C 180,E1 -4939.237,E2 -4939.237} C_VEL
LIN {X 0,Y 517.132,Z 473.999,A -85,B 0,C 180,E1 -4940.22,E2 -4940.22} C_VEL
LIN {X 0,Y 516.865,Z 483.293,A -85,B 0,C 180,E1 -4941.399,E2 -4941.399} C_VEL
LIN {X 0,Y 516.641,Z 490.69,A -85,B 0,C 180,E1 -4942.576,E2 -4942.576} C_VEL
LIN {X 0,Y 516.552,Z 496.628,A -85,B 0,C 180,E1 -4943.752,E2 -4943.752} C_VEL
LIN {X 0,Y 516.32,Z 501.333,A -85,B 0,C 180,E1 -4944.925,E2 -4944.925} C_VEL
LIN {X 0,Y 516.373,Z 504.923,A -85,B 0,C 180,E1 -4946.099,E2 -4946.099} C_VEL
LIN {X 0,Y 516.382,Z 506.772,A -85,B 0,C 180,E1 -4946.88,E2 -4946.88} C_VEL
LIN {X 0,Y 516.267,Z 508.196,A -85,B 0,C 180,E1 -4947.66,E2 -4947.66} C_VEL
LIN {X 0,Y 516.168,Z 509.807,A -85,B 0,C 180,E1 -4949.221,E2 -4949.221} C_VEL
LIN {X 0,Y 516.167,Z 510.044,A -85,B 0,C 180,E1 -4950.001,E2 -4950.001} C_VEL
LIN {X 0,Y 516.168,Z 509.86,A -85,B 0,C 180,E1 -4950.781,E2 -4950.781} C_VEL
LIN {X 0,Y 516.267,Z 508.321,A -85,B 0,C 180,E1 -4952.341,E2 -4952.341} C_VEL
LIN {X 0,Y 516.383,Z 506.966,A -85,B 0,C 180,E1 -4953.121,E2 -4953.121} C_VEL
LIN {X 0,Y 516.374,Z 504.122,A -85,B 0,C 180,E1 -4954.294,E2 -4954.294} C_VEL
LIN {X 0,Y 516.407,Z 500.255,A -85,B 0,C 180,E1 -4955.467,E2 -4955.467} C_VEL
LIN {X 0,Y 516.548,Z 494.315,A -85,B 0,C 180,E1 -4956.829,E2 -4956.829} C_VEL
LIN {X 0,Y 516.737,Z 487.738,A -85,B 0,C 180,E1 -4958.014,E2 -4958.014} C_VEL
LIN {X 0,Y 516.946,Z 479.607,A -85,B 0,C 180,E1 -4959.193,E2 -4959.193} C_VEL
LIN {X 0,Y 517.205,Z 471.227,A -85,B 0,C 180,E1 -4960.175,E2 -4960.175} C_VEL
LIN {X 0,Y 517.514,Z 460.955,A -85,B 0,C 180,E1 -4961.159,E2 -4961.159} C_VEL
LIN {X 0,Y 517.812,Z 450.725,A -85,B 0,C 180,E1 -4961.951,E2 -4961.951} C_VEL
LIN {X 0,Y 518.094,Z 439.549,A -85,B 0,C 180,E1 -4962.636,E2 -4962.636} C_VEL
LIN {X 0,Y 518.349,Z 426.905,A -85,B 0,C 180,E1 -4963.227,E2 -4963.227} C_VEL
LIN {X 0,Y 518.59,Z 414.357,A -85,B 0,C 180,E1 -4963.645,E2 -4963.645} C_VEL
LIN {X 0,Y 518.725,Z 401.254,A -85,B 0,C 180,E1 -4963.916,E2 -4963.916} C_VEL
LIN {X 0,Y 519.056,Z 309.629,A -85,B 0,C 180,E1 -4965.193,E2 -4965.193} C_VEL
LIN {X 0,Y 516.864,Z 296.003,A -85,B 0,C 180,E1 -4965.462,E2 -4965.462} C_VEL
LIN {X 0,Y 516.776,Z 285.298,A -85,B 0,C 180,E1 -4966.798,E2 -4966.798} C_VEL
LIN {X 0,Y 516.792,Z 281.116,A -85,B 0,C 180,E1 -4967.409,E2 -4967.409} C_VEL
LIN {X 0,Y 516.926,Z 281.096,A -85,B 0,C 180,E1 -4969.045,E2 -4969.045} C_VEL
LIN {X 0,Y 516.891,Z 281.102,A -85,B 0,C 180,E1 -4971.538,E2 -4971.538} C_VEL
LIN {X 0,Y 516.89,Z 281.096,A -85,B 0,C 180,E1 -4974.358,E2 -4974.358} C_VEL
LIN {X 0,Y 516.927,Z 281.092,A -85,B 0,C 180,E1 -4976.658,E2 -4976.658} C_VEL
LIN {X 0,Y 516.914,Z 281.098,A -85,B 0,C 180,E1 -4979.524,E2 -4979.524} C_VEL
LIN {X 0,Y 516.899,Z 281.095,A -85,B 0,C 180,E1 -4982.543,E2 -4982.543} C_VEL
LIN {X 0,Y 516.87,Z 281.105,A -85,B 0,C 180,E1 -4985.33,E2 -4985.33} C_VEL
LIN {X 0,Y 516.884,Z 281.096,A -85,B 0,C 180,E1 -4987.943,E2 -4987.943} C_VEL
LIN {X 0,Y 516.888,Z 281.099,A -85,B 0,C 180,E1 -4990.742,E2 -4990.742} C_VEL
LIN {X 0,Y 516.889,Z 281.099,A -85,B 0,C 180,E1 -4992.832,E2 -4992.832} C_VEL
LIN {X 0,Y 516.928,Z 281.097,A -85,B 0,C 180,E1 -4995.01,E2 -4995.01} C_VEL
LIN {X 0,Y 516.918,Z 281.093,A -85,B 0,C 180,E1 -4998.399,E2 -4998.399} C_VEL
LIN {X 0,Y 516.887,Z 281.099,A -85,B 0,C 180,E1 -5001.284,E2 -5001.284} C_VEL
LIN {X 0,Y 516.876,Z 281.098,A -85,B 0,C 180,E1 -5004.22,E2 -5004.22} C_VEL
LIN {X 0,Y 516.9,Z 281.099,A -85,B 0,C 180,E1 -5007.053,E2 -5007.053} C_VEL
LIN {X 0,Y 516.896,Z 281.094,A -85,B 0,C 180,E1 -5009.796,E2 -5009.796} C_VEL
LIN {X 0,Y 516.927,Z 281.094,A -85,B 0,C 180,E1 -5012.467,E2 -5012.467} C_VEL
LIN {X 0,Y 516.89,Z 281.094,A -85,B 0,C 180,E1 -5015.642,E2 -5015.642} C_VEL
LIN {X 0,Y 516.89,Z 281.101,A -85,B 0,C 180,E1 -5018.462,E2 -5018.462} C_VEL
LIN {X 0,Y 516.968,Z 281.253,A -85,B 0,C 180,E1 -5020.803,E2 -5020.803} C_VEL
LIN {X 0,Y 517.475,Z 286.583,A -85,B 0,C 180,E1 -5021.934,E2 -5021.934} C_VEL
LIN {X 0,Y 517.204,Z 300.061,A -85,B 0,C 180,E1 -5024.702,E2 -5024.702} C_VEL
LIN {X 0,Y 519.078,Z 310.285,A -85,B 0,C 180,E1 -5024.925,E2 -5024.925} C_VEL
LIN {X 0,Y 518.457,Z 407.046,A -85,B 0,C 180,E1 -5026.352,E2 -5026.352} C_VEL
LIN {X 0,Y 518.332,Z 420.77,A -85,B 0,C 180,E1 -5026.723,E2 -5026.723} C_VEL
LIN {X 0,Y 518.056,Z 433.12,A -85,B 0,C 180,E1 -5027.215,E2 -5027.215} C_VEL
LIN {X 0,Y 517.815,Z 445.158,A -85,B 0,C 180,E1 -5027.865,E2 -5027.865} C_VEL
LIN {X 0,Y 517.568,Z 456.405,A -85,B 0,C 180,E1 -5028.645,E2 -5028.645} C_VEL
LIN {X 0,Y 517.242,Z 466.651,A -85,B 0,C 180,E1 -5029.529,E2 -5029.529} C_VEL
LIN {X 0,Y 517.02,Z 475.032,A -85,B 0,C 180,E1 -5030.415,E2 -5030.415} C_VEL
LIN {X 0,Y 516.77,Z 484.136,A -85,B 0,C 180,E1 -5031.593,E2 -5031.593} C_VEL
LIN {X 0,Y 516.614,Z 491.45,A -85,B 0,C 180,E1 -5032.771,E2 -5032.771} C_VEL
LIN {X 0,Y 516.495,Z 498.113,A -85,B 0,C 180,E1 -5034.143,E2 -5034.143} C_VEL
LIN {X 0,Y 516.323,Z 502.511,A -85,B 0,C 180,E1 -5035.315,E2 -5035.315} C_VEL
LIN {X 0,Y 516.375,Z 504.854,A -85,B 0,C 180,E1 -5036.098,E2 -5036.098} C_VEL
LIN {X 0,Y 516.383,Z 506.726,A -85,B 0,C 180,E1 -5036.879,E2 -5036.879} C_VEL
LIN {X 0,Y 516.193,Z 509.214,A -85,B 0,C 180,E1 -5038.44,E2 -5038.44} C_VEL
LIN {X 0,Y 516.17,Z 509.84,A -85,B 0,C 180,E1 -5039.22,E2 -5039.22} C_VEL
LIN {X 0,Y 516.171,Z 510.071,A -85,B 0,C 180,E1 -5040,E2 -5040} C_VEL
LIN {X 0,Y 516.169,Z 509.912,A -85,B 0,C 180,E1 -5040.78,E2 -5040.78} C_VEL
LIN {X 0,Y 516.193,Z 509.338,A -85,B 0,C 180,E1 -5041.56,E2 -5041.56} C_VEL
LIN {X 0,Y 516.384,Z 506.993,A -85,B 0,C 180,E1 -5043.121,E2 -5043.121} C_VEL
LIN {X 0,Y 516.374,Z 504.108,A -85,B 0,C 180,E1 -5044.293,E2 -5044.293} C_VEL
LIN {X 0,Y 516.406,Z 500.179,A -85,B 0,C 180,E1 -5045.467,E2 -5045.467} C_VEL
LIN {X 0,Y 516.546,Z 494.156,A -85,B 0,C 180,E1 -5046.827,E2 -5046.827} C_VEL
LIN {X 0,Y 516.682,Z 487.447,A -85,B 0,C 180,E1 -5048.014,E2 -5048.014} C_VEL
LIN {X 0,Y 516.917,Z 479.158,A -85,B 0,C 180,E1 -5049.193,E2 -5049.193} C_VEL
LIN {X 0,Y 517.16,Z 470.6,A -85,B 0,C 180,E1 -5050.176,E2 -5050.176} C_VEL
LIN {X 0,Y 517.428,Z 461.185,A -85,B 0,C 180,E1 -5051.061,E2 -5051.061} C_VEL
LIN {X 0,Y 517.706,Z 450.274,A -85,B 0,C 180,E1 -5051.893,E2 -5051.893} C_VEL
LIN {X 0,Y 517.933,Z 439.644,A -85,B 0,C 180,E1 -5052.539,E2 -5052.539} C_VEL
LIN {X 0,Y 518.164,Z 428.183,A -85,B 0,C 180,E1 -5053.082,E2 -5053.082} C_VEL
LIN {X 0,Y 518.389,Z 415.062,A -85,B 0,C 180,E1 -5053.525,E2 -5053.525} C_VEL
LIN {X 0,Y 518.487,Z 402.525,A -85,B 0,C 180,E1 -5053.797,E2 -5053.797} C_VEL
LIN {X 0,Y 519.076,Z 310.055,A -85,B 0,C 180,E1 -5055.166,E2 -5055.166} C_VEL
LIN {X 0,Y 517.335,Z 301.021,A -85,B 0,C 180,E1 -5055.372,E2 -5055.372} C_VEL
LIN {X 0,Y 517.669,Z 287.596,A -85,B 0,C 180,E1 -5058.195,E2 -5058.195} C_VEL
LIN {X 0,Y 516.952,Z 281.095,A -85,B 0,C 180,E1 -5059.662,E2 -5059.662} C_VEL
LIN {X 0,Y 516.867,Z 281.101,A -85,B 0,C 180,E1 -5062.388,E2 -5062.388} C_VEL
LIN {X 0,Y 516.838,Z 281.108,A -85,B 0,C 180,E1 -5064.932,E2 -5064.932} C_VEL
LIN {X 0,Y 516.858,Z 281.102,A -85,B 0,C 180,E1 -5067.89,E2 -5067.89} C_VEL
LIN {X 0,Y 516.851,Z 281.108,A -85,B 0,C 180,E1 -5071.112,E2 -5071.112} C_VEL
LIN {X 0,Y 516.87,Z 281.099,A -85,B 0,C 180,E1 -5073.959,E2 -5073.959} C_VEL
LIN {X 0,Y 516.8,Z 281.114,A -85,B 0,C 180,E1 -5076.753,E2 -5076.753} C_VEL
LIN {X 0,Y 516.857,Z 281.099,A -85,B 0,C 180,E1 -5079.724,E2 -5079.724} C_VEL
LIN {X 0,Y 516.844,Z 281.107,A -85,B 0,C 180,E1 -5082.836,E2 -5082.836} C_VEL
LIN {X 0,Y 516.9,Z 281.097,A -85,B 0,C 180,E1 -5085.007,E2 -5085.007} C_VEL
LIN {X 0,Y 516.851,Z 281.107,A -85,B 0,C 180,E1 -5088.407,E2 -5088.407} C_VEL
LIN {X 0,Y 516.878,Z 281.097,A -85,B 0,C 180,E1 -5091.283,E2 -5091.283} C_VEL
LIN {X 0,Y 516.87,Z 281.106,A -85,B 0,C 180,E1 -5094.219,E2 -5094.219} C_VEL
LIN {X 0,Y 516.892,Z 281.098,A -85,B 0,C 180,E1 -5097.052,E2 -5097.052} C_VEL
LIN {X 0,Y 516.887,Z 281.105,A -85,B 0,C 180,E1 -5099.795,E2 -5099.795} C_VEL
LIN {X 0,Y 516.897,Z 281.1,A -85,B 0,C 180,E1 -5102.465,E2 -5102.465} C_VEL
LIN {X 0,Y 516.963,Z 281.282,A -85,B 0,C 180,E1 -5104.859,E2 -5104.859} C_VEL
LIN {X 0,Y 518.436,Z 289.263,A -85,B 0,C 180,E1 -5106.215,E2 -5106.215} C_VEL
LIN {X 0,Y 518.319,Z 298.642,A -85,B 0,C 180,E1 -5107.687,E2 -5107.687} C_VEL
LIN {X 0,Y 517.773,Z 317.452,A -85,B 0,C 180,E1 -5110.576,E2 -5110.576} C_VEL
LIN {X 0,Y 517.408,Z 335.023,A -85,B 0,C 180,E1 -5113.223,E2 -5113.223} C_VEL
LIN {X 0,Y 517.254,Z 344.469,A -85,B 0,C 180,E1 -5114.631,E2 -5114.631} C_VEL
LIN {X 0,Y 518.98,Z 357.775,A -85,B 0,C 180,E1 -5114.9,E2 -5114.9} C_VEL
LIN {X 0,Y 518.399,Z 454.135,A -85,B 0,C 180,E1 -5116.325,E2 -5116.325} C_VEL
LIN {X 0,Y 518.137,Z 467.869,A -85,B 0,C 180,E1 -5116.693,E2 -5116.693} C_VEL
LIN {X 0,Y 517.896,Z 480.819,A -85,B 0,C 180,E1 -5117.21,E2 -5117.21} C_VEL
LIN {X 0,Y 517.652,Z 492.325,A -85,B 0,C 180,E1 -5117.83,E2 -5117.83} C_VEL
LIN {X 0,Y 517.317,Z 504.121,A -85,B 0,C 180,E1 -5118.638,E2 -5118.638} C_VEL
LIN {X 0,Y 517.091,Z 514.425,A -85,B 0,C 180,E1 -5119.526,E2 -5119.526} C_VEL
LIN {X 0,Y 516.795,Z 524.517,A -85,B 0,C 180,E1 -5120.607,E2 -5120.607} C_VEL
LIN {X 0,Y 516.61,Z 533.412,A -85,B 0,C 180,E1 -5121.787,E2 -5121.787} C_VEL
LIN {X 0,Y 516.442,Z 540.481,A -85,B 0,C 180,E1 -5122.964,E2 -5122.964} C_VEL
LIN {X 0,Y 516.417,Z 546.14,A -85,B 0,C 180,E1 -5124.141,E2 -5124.141} C_VEL
LIN {X 0,Y 516.27,Z 550.574,A -85,B 0,C 180,E1 -5125.314,E2 -5125.314} C_VEL
LIN {X 0,Y 516.37,Z 552.928,A -85,B 0,C 180,E1 -5126.097,E2 -5126.097} C_VEL
LIN {X 0,Y 516.282,Z 554.836,A -85,B 0,C 180,E1 -5126.878,E2 -5126.878} C_VEL
LIN {X 0,Y 516.261,Z 556.263,A -85,B 0,C 180,E1 -5127.659,E2 -5127.659} C_VEL
LIN {X 0,Y 516.163,Z 557.902,A -85,B 0,C 180,E1 -5129.219,E2 -5129.219} C_VEL
LIN {X 0,Y 516.162,Z 558.131,A -85,B 0,C 180,E1 -5129.999,E2 -5129.999} C_VEL
LIN {X 0,Y 516.162,Z 557.916,A -85,B 0,C 180,E1 -5130.779,E2 -5130.779} C_VEL
LIN {X 0,Y 516.261,Z 556.303,A -85,B 0,C 180,E1 -5132.34,E2 -5132.34} C_VEL
LIN {X 0,Y 516.282,Z 554.888,A -85,B 0,C 180,E1 -5133.121,E2 -5133.121} C_VEL
LIN {X 0,Y 516.312,Z 551.919,A -85,B 0,C 180,E1 -5134.293,E2 -5134.293} C_VEL
LIN {X 0,Y 516.396,Z 547.893,A -85,B 0,C 180,E1 -5135.466,E2 -5135.466} C_VEL
LIN {X 0,Y 516.451,Z 541.882,A -85,B 0,C 180,E1 -5136.799,E2 -5136.799} C_VEL
LIN {X 0,Y 516.583,Z 534.895,A -85,B 0,C 180,E1 -5138.015,E2 -5138.015} C_VEL
LIN {X 0,Y 516.769,Z 526.463,A -85,B 0,C 180,E1 -5139.194,E2 -5139.194} C_VEL
LIN {X 0,Y 516.967,Z 517.772,A -85,B 0,C 180,E1 -5140.179,E2 -5140.179} C_VEL
LIN {X 0,Y 517.353,Z 507.071,A -85,B 0,C 180,E1 -5141.161,E2 -5141.161} C_VEL
LIN {X 0,Y 517.548,Z 497.52,A -85,B 0,C 180,E1 -5141.876,E2 -5141.876} C_VEL
LIN {X 0,Y 517.827,Z 486.527,A -85,B 0,C 180,E1 -5142.541,E2 -5142.541} C_VEL
LIN {X 0,Y 518.098,Z 474.996,A -85,B 0,C 180,E1 -5143.082,E2 -5143.082} C_VEL
LIN {X 0,Y 518.3,Z 461.77,A -85,B 0,C 180,E1 -5143.526,E2 -5143.526} C_VEL
LIN {X 0,Y 518.551,Z 449.167,A -85,B 0,C 180,E1 -5143.794,E2 -5143.794} C_VEL
LIN {X 0,Y 518.939,Z 371.202,A -85,B 0,C 180,E1 -5144.91,E2 -5144.91} C_VEL
LIN {X 0,Y 518.94,Z 356.375,A -85,B 0,C 180,E1 -5145.133,E2 -5145.133} C_VEL
LIN {X 0,Y 517.325,Z 345.311,A -85,B 0,C 180,E1 -5145.358,E2 -5145.358} C_VEL
LIN {X 0,Y 517.754,Z 325.285,A -85,B 0,C 180,E1 -5148.396,E2 -5148.396} C_VEL
LIN {X 0,Y 518.236,Z 307.798,A -85,B 0,C 180,E1 -5151.061,E2 -5151.061} C_VEL
LIN {X 0,Y 518.717,Z 290.387,A -85,B 0,C 180,E1 -5153.77,E2 -5153.77} C_VEL
LIN {X 0,Y 516.956,Z 281.093,A -85,B 0,C 180,E1 -5155.355,E2 -5155.355} C_VEL
LIN {X 0,Y 516.907,Z 281.098,A -85,B 0,C 180,E1 -5158.415,E2 -5158.415} C_VEL
LIN {X 0,Y 516.886,Z 281.095,A -85,B 0,C 180,E1 -5161.109,E2 -5161.109} C_VEL
LIN {X 0,Y 516.904,Z 281.101,A -85,B 0,C 180,E1 -5163.965,E2 -5163.965} C_VEL
LIN {X 0,Y 516.849,Z 281.1,A -85,B 0,C 180,E1 -5166.747,E2 -5166.747} C_VEL
LIN {X 0,Y 516.877,Z 281.103,A -85,B 0,C 180,E1 -5169.72,E2 -5169.72} C_VEL
LIN {X 0,Y 516.9,Z 281.102,A -85,B 0,C 180,E1 -5171.775,E2 -5171.775} C_VEL
LIN {X 0,Y 516.89,Z 281.096,A -85,B 0,C 180,E1 -5175.006,E2 -5175.006} C_VEL
LIN {X 0,Y 516.896,Z 281.094,A -85,B 0,C 180,E1 -5178.399,E2 -5178.399} C_VEL
LIN {X 0,Y 516.87,Z 281.102,A -85,B 0,C 180,E1 -5181.283,E2 -5181.283} C_VEL
LIN {X 0,Y 516.863,Z 281.099,A -85,B 0,C 180,E1 -5184.219,E2 -5184.219} C_VEL
LIN {X 0,Y 516.873,Z 281.101,A -85,B 0,C 180,E1 -5187.051,E2 -5187.051} C_VEL
LIN {X 0,Y 516.858,Z 281.101,A -85,B 0,C 180,E1 -5189.794,E2 -5189.794} C_VEL
LIN {X 0,Y 516.867,Z 281.099,A -85,B 0,C 180,E1 -5192.464,E2 -5192.464} C_VEL
LIN {X 0,Y 516.835,Z 281.108,A -85,B 0,C 180,E1 -5195.068,E2 -5195.068} C_VEL
LIN {X 0,Y 516.86,Z 281.101,A -85,B 0,C 180,E1 -5197.621,E2 -5197.621} C_VEL
LIN {X 0,Y 516.92,Z 281.092,A -85,B 0,C 180,E1 -5200.129,E2 -5200.129} C_VEL
LIN {X 0,Y 516.884,Z 281.1,A -85,B 0,C 180,E1 -5202.595,E2 -5202.595} C_VEL
LIN {X 0,Y 516.921,Z 281.098,A -85,B 0,C 180,E1 -5205.029,E2 -5205.029} C_VEL
LIN {X 0,Y 516.957,Z 281.09,A -85,B 0,C 180,E1 -5208.233,E2 -5208.233} C_VEL
LIN {X 0,Y 516.939,Z 281.091,A -85,B 0,C 180,E1 -5211.399,E2 -5211.399} C_VEL
LIN {X 0,Y 516.969,Z 281.091,A -85,B 0,C 180,E1 -5214.539,E2 -5214.539} C_VEL
LIN {X 0,Y 517.059,Z 281.075,A -85,B 0,C 180,E1 -5217.663,E2 -5217.663} C_VEL
LIN {X 0,Y 517.078,Z 281.077,A -85,B 0,C 180,E1 -5220.779,E2 -5220.779} C_VEL
LIN {X 0,Y 516.931,Z 281.092,A -85,B 0,C 180,E1 -5223.117,E2 -5223.117} C_VEL
LIN {X 0,Y 516.96,Z 281.092,A -85,B 0,C 180,E1 -5226.244,E2 -5226.244} C_VEL
LIN {X 0,Y 516.923,Z 281.092,A -85,B 0,C 180,E1 -5229.39,E2 -5229.39} C_VEL
LIN {X 0,Y 516.943,Z 281.094,A -85,B 0,C 180,E1 -5231.807,E2 -5231.807} C_VEL
LIN {X 0,Y 516.93,Z 281.091,A -85,B 0,C 180,E1 -5235.144,E2 -5235.144} C_VEL
LIN {X 0,Y 516.903,Z 281.1,A -85,B 0,C 180,E1 -5238.223,E2 -5238.223} C_VEL
LIN {X 0,Y 516.896,Z 281.096,A -85,B 0,C 180,E1 -5240.702,E2 -5240.702} C_VEL
LIN {X 0,Y 516.882,Z 281.102,A -85,B 0,C 180,E1 -5244.074,E2 -5244.074} C_VEL
LIN {X 0,Y 516.882,Z 281.098,A -85,B 0,C 180,E1 -5246.66,E2 -5246.66} C_VEL
LIN {X 0,Y 516.901,Z 281.099,A -85,B 0,C 180,E1 -5249.524,E2 -5249.524} C_VEL
LIN {X 0,Y 516.888,Z 281.097,A -85,B 0,C 180,E1 -5252.544,E2 -5252.544} C_VEL
LIN {X 0,Y 516.857,Z 281.105,A -85,B 0,C 180,E1 -5255.33,E2 -5255.33} C_VEL
LIN {X 0,Y 516.872,Z 281.101,A -85,B 0,C 180,E1 -5257.943,E2 -5257.943} C_VEL
LIN {X 0,Y 516.876,Z 281.099,A -85,B 0,C 180,E1 -5260.743,E2 -5260.743} C_VEL
LIN {X 0,Y 516.876,Z 281.1,A -85,B 0,C 180,E1 -5263.904,E2 -5263.904} C_VEL
LIN {X 0,Y 516.861,Z 281.101,A -85,B 0,C 180,E1 -5266.911,E2 -5266.911} C_VEL
LIN {X 0,Y 516.88,Z 281.101,A -85,B 0,C 180,E1 -5269.591,E2 -5269.591} C_VEL
LIN {X 0,Y 516.877,Z 281.098,A -85,B 0,C 180,E1 -5270.296,E2 -5270.296} C_VEL
LIN {X 0,Y 516.206,Z 281.187,A -85,B 0,C 180,E1 -5270.946,E2 -5270.946} C_VEL
LIN {X 0,Y 513.359,Z 281.542,A -85,B 0,C 180,E1 -5272.002,E2 -5272.002} C_VEL
LIN {X 0,Y 510.95,Z 281.842,A -85,B 0,C 180,E1 -5272.852,E2 -5272.852} C_VEL
LIN {X 0,Y 509.907,Z 281.969,A -85,B 0,C 180,E1 -5273.509,E2 -5273.509} C_VEL
LIN {X 0,Y 509.817,Z 281.979,A -85,B 0,C 180,E1 -5273.731,E2 -5273.731} C_VEL
LIN {X 0,Y 509.839,Z 281.978,A -85,B 0,C 180,E1 -5276.539,E2 -5276.539} C_VEL
LIN {X 0,Y 509.84,Z 281.978,A -85,B 0,C 180,E1 -5279.335,E2 -5279.335} C_VEL
LIN {X 0,Y 509.884,Z 281.97,A -85,B 0,C 180,E1 -5282.055,E2 -5282.055} C_VEL
LIN {X 0,Y 509.872,Z 281.975,A -85,B 0,C 180,E1 -5284.705,E2 -5284.705} C_VEL
LIN {X 0,Y 509.826,Z 281.977,A -85,B 0,C 180,E1 -5287.459,E2 -5287.459} C_VEL
LIN {X 0,Y 509.918,Z 281.965,A -85,B 0,C 180,E1 -5289.846,E2 -5289.846} C_VEL
LIN {X 0,Y 509.887,Z 281.977,A -85,B 0,C 180,E1 -5292.349,E2 -5292.349} C_VEL
LIN {X 0,Y 509.705,Z 282.164,A -85,B 0,C 180,E1 -5292.834,E2 -5292.834} C_VEL
LIN {X 0,Y 509.706,Z 291.622,A -85,B 0,C 180,E1 -5293.993,E2 -5293.993} C_VEL
LIN {X 0,Y 509.858,Z 295.805,A -85,B 0,C 180,E1 -5294.414,E2 -5294.414} C_VEL
LIN {X 0,Y 512.292,Z 312.061,A -85,B 0,C 180,E1 -5294.724,E2 -5294.724} C_VEL
LIN {X 0,Y 511.795,Z 406.375,A -85,B 0,C 180,E1 -5296.071,E2 -5296.071} C_VEL
LIN {X 0,Y 511.599,Z 419.994,A -85,B 0,C 180,E1 -5296.42,E2 -5296.42} C_VEL
LIN {X 0,Y 511.302,Z 432.113,A -85,B 0,C 180,E1 -5296.892,E2 -5296.892} C_VEL
LIN {X 0,Y 511.07,Z 443.934,A -85,B 0,C 180,E1 -5297.518,E2 -5297.518} C_VEL
LIN {X 0,Y 510.779,Z 455.317,A -85,B 0,C 180,E1 -5298.291,E2 -5298.291} C_VEL
LIN {X 0,Y 510.405,Z 465.759,A -85,B 0,C 180,E1 -5299.188,E2 -5299.188} C_VEL
LIN {X 0,Y 510.108,Z 476.026,A -85,B 0,C 180,E1 -5300.284,E2 -5300.284} C_VEL
LIN {X 0,Y 509.811,Z 484.931,A -85,B 0,C 180,E1 -5301.479,E2 -5301.479} C_VEL
LIN {X 0,Y 509.574,Z 492.086,A -85,B 0,C 180,E1 -5302.671,E2 -5302.671} C_VEL
LIN {X 0,Y 509.497,Z 496.944,A -85,B 0,C 180,E1 -5303.665,E2 -5303.665} C_VEL
LIN {X 0,Y 509.254,Z 501.649,A -85,B 0,C 180,E1 -5304.854,E2 -5304.854} C_VEL
LIN {X 0,Y 509.306,Z 505.239,A -85,B 0,C 180,E1 -5306.045,E2 -5306.045} C_VEL
LIN {X 0,Y 509.305,Z 507.09,A -85,B 0,C 180,E1 -5306.837,E2 -5306.837} C_VEL
LIN {X 0,Y 509.199,Z 508.513,A -85,B 0,C 180,E1 -5307.628,E2 -5307.628} C_VEL
LIN {X 0,Y 509.081,Z 510.124,A -85,B 0,C 180,E1 -5309.21,E2 -5309.21} C_VEL
LIN {X 0,Y 509.077,Z 510.361,A -85,B 0,C 180,E1 -5310.001,E2 -5310.001} C_VEL
LIN {X 0,Y 509.081,Z 510.176,A -85,B 0,C 180,E1 -5310.792,E2 -5310.792} C_VEL
LIN {X 0,Y 509.199,Z 508.636,A -85,B 0,C 180,E1 -5312.374,E2 -5312.374} C_VEL
LIN {X 0,Y 509.305,Z 507.281,A -85,B 0,C 180,E1 -5313.165,E2 -5313.165} C_VEL
LIN {X 0,Y 509.301,Z 504.436,A -85,B 0,C 180,E1 -5314.353,E2 -5314.353} C_VEL
LIN {X 0,Y 509.352,Z 500.566,A -85,B 0,C 180,E1 -5315.543,E2 -5315.543} C_VEL
LIN {X 0,Y 509.471,Z 495.428,A -85,B 0,C 180,E1 -5316.761,E2 -5316.761} C_VEL
LIN {X 0,Y 509.694,Z 488.045,A -85,B 0,C 180,E1 -5318.126,E2 -5318.126} C_VEL
LIN {X 0,Y 509.943,Z 479.909,A -85,B 0,C 180,E1 -5319.32,E2 -5319.32} C_VEL
LIN {X 0,Y 510.206,Z 471.525,A -85,B 0,C 180,E1 -5320.316,E2 -5320.316} C_VEL
LIN {X 0,Y 510.545,Z 461.245,A -85,B 0,C 180,E1 -5321.313,E2 -5321.313} C_VEL
LIN {X 0,Y 510.922,Z 450.14,A -85,B 0,C 180,E1 -5322.174,E2 -5322.174} C_VEL
LIN {X 0,Y 511.206,Z 437.942,A -85,B 0,C 180,E1 -5322.91,E2 -5322.91} C_VEL
LIN {X 0,Y 511.496,Z 425.937,A -85,B 0,C 180,E1 -5323.458,E2 -5323.458} C_VEL
LIN {X 0,Y 511.68,Z 412.549,A -85,B 0,C 180,E1 -5323.883,E2 -5323.883} C_VEL
LIN {X 0,Y 511.913,Z 399.566,A -85,B 0,C 180,E1 -5324.13,E2 -5324.13} C_VEL
LIN {X 0,Y 512.163,Z 310.18,A -85,B 0,C 180,E1 -5325.397,E2 -5325.397} C_VEL
LIN {X 0,Y 509.809,Z 295.2,A -85,B 0,C 180,E1 -5325.71,E2 -5325.71} C_VEL
LIN {X 0,Y 509.682,Z 285.453,A -85,B 0,C 180,E1 -5326.833,E2 -5326.833} C_VEL
LIN {X 0,Y 509.681,Z 282.002,A -85,B 0,C 180,E1 -5327.298,E2 -5327.298} C_VEL
LIN {X 0,Y 509.882,Z 281.972,A -85,B 0,C 180,E1 -5328.484,E2 -5328.484} C_VEL
LIN {X 0,Y 509.856,Z 281.975,A -85,B 0,C 180,E1 -5331.002,E2 -5331.002} C_VEL
LIN {X 0,Y 509.828,Z 281.982,A -85,B 0,C 180,E1 -5333.564,E2 -5333.564} C_VEL
LIN {X 0,Y 509.915,Z 281.965,A -85,B 0,C 180,E1 -5336.378,E2 -5336.378} C_VEL
LIN {X 0,Y 509.877,Z 281.972,A -85,B 0,C 180,E1 -5338.845,E2 -5338.845} C_VEL
LIN {X 0,Y 509.824,Z 281.98,A -85,B 0,C 180,E1 -5341.591,E2 -5341.591} C_VEL
LIN {X 0,Y 509.843,Z 281.974,A -85,B 0,C 180,E1 -5344.415,E2 -5344.415} C_VEL
LIN {X 0,Y 509.821,Z 281.983,A -85,B 0,C 180,E1 -5347.341,E2 -5347.341} C_VEL
LIN {X 0,Y 509.843,Z 281.974,A -85,B 0,C 180,E1 -5350.382,E2 -5350.382} C_VEL
LIN {X 0,Y 509.829,Z 281.981,A -85,B 0,C 180,E1 -5353.063,E2 -5353.063} C_VEL
LIN {X 0,Y 509.835,Z 281.974,A -85,B 0,C 180,E1 -5355.793,E2 -5355.793} C_VEL
LIN {X 0,Y 509.86,Z 281.973,A -85,B 0,C 180,E1 -5358.575,E2 -5358.575} C_VEL
LIN {X 0,Y 509.856,Z 281.971,A -85,B 0,C 180,E1 -5361.787,E2 -5361.787} C_VEL
LIN {X 0,Y 509.834,Z 281.978,A -85,B 0,C 180,E1 -5364.622,E2 -5364.622} C_VEL
LIN {X 0,Y 509.866,Z 281.971,A -85,B 0,C 180,E1 -5367.481,E2 -5367.481} C_VEL
LIN {X 0,Y 509.863,Z 281.972,A -85,B 0,C 180,E1 -5370.274,E2 -5370.274} C_VEL
LIN {X 0,Y 509.879,Z 281.974,A -85,B 0,C 180,E1 -5372.944,E2 -5372.944} C_VEL
LIN {X 0,Y 509.854,Z 281.971,A -85,B 0,C 180,E1 -5375.573,E2 -5375.573} C_VEL
LIN {X 0,Y 509.826,Z 281.977,A -85,B 0,C 180,E1 -5378.149,E2 -5378.149} C_VEL
LIN {X 0,Y 509.937,Z 282.065,A -85,B 0,C 180,E1 -5380.658,E2 -5380.658} C_VEL
LIN {X 0,Y 510.488,Z 287.357,A -85,B 0,C 180,E1 -5381.795,E2 -5381.795} C_VEL
LIN {X 0,Y 510.205,Z 300.347,A -85,B 0,C 180,E1 -5384.493,E2 -5384.493} C_VEL
LIN {X 0,Y 512.219,Z 310.867,A -85,B 0,C 180,E1 -5384.726,E2 -5384.726} C_VEL
LIN {X 0,Y 511.54,Z 407.637,A -85,B 0,C 180,E1 -5386.189,E2 -5386.189} C_VEL
LIN {X 0,Y 511.41,Z 421.242,A -85,B 0,C 180,E1 -5386.565,E2 -5386.565} C_VEL
LIN {X 0,Y 511.103,Z 433.016,A -85,B 0,C 180,E1 -5387.038,E2 -5387.038} C_VEL
LIN {X 0,Y 510.894,Z 444.897,A -85,B 0,C 180,E1 -5387.683,E2 -5387.683} C_VEL
LIN {X 0,Y 510.601,Z 456.447,A -85,B 0,C 180,E1 -5388.487,E2 -5388.487} C_VEL
LIN {X 0,Y 510.267,Z 466.777,A -85,B 0,C 180,E1 -5389.384,E2 -5389.384} C_VEL
LIN {X 0,Y 509.962,Z 476.848,A -85,B 0,C 180,E1 -5390.481,E2 -5390.481} C_VEL
LIN {X 0,Y 509.707,Z 485.693,A -85,B 0,C 180,E1 -5391.676,E2 -5391.676} C_VEL
LIN {X 0,Y 509.529,Z 492.752,A -85,B 0,C 180,E1 -5392.869,E2 -5392.869} C_VEL
LIN {X 0,Y 509.437,Z 498.381,A -85,B 0,C 180,E1 -5394.061,E2 -5394.061} C_VEL
LIN {X 0,Y 509.239,Z 502.806,A -85,B 0,C 180,E1 -5395.25,E2 -5395.25} C_VEL
LIN {X 0,Y 509.307,Z 505.141,A -85,B 0,C 180,E1 -5396.044,E2 -5396.044} C_VEL
LIN {X 0,Y 509.305,Z 507.04,A -85,B 0,C 180,E1 -5396.836,E2 -5396.836} C_VEL
LIN {X 0,Y 509.198,Z 508.494,A -85,B 0,C 180,E1 -5397.627,E2 -5397.627} C_VEL
LIN {X 0,Y 509.083,Z 510.169,A -85,B 0,C 180,E1 -5399.209,E2 -5399.209} C_VEL
LIN {X 0,Y 509.081,Z 510.421,A -85,B 0,C 180,E1 -5400,E2 -5400} C_VEL
LIN {X 0,Y 509.082,Z 510.245,A -85,B 0,C 180,E1 -5400.791,E2 -5400.791} C_VEL
LIN {X 0,Y 509.198,Z 508.69,A -85,B 0,C 180,E1 -5402.373,E2 -5402.373} C_VEL
LIN {X 0,Y 509.306,Z 507.318,A -85,B 0,C 180,E1 -5403.164,E2 -5403.164} C_VEL
LIN {X 0,Y 509.301,Z 504.419,A -85,B 0,C 180,E1 -5404.353,E2 -5404.353} C_VEL
LIN {X 0,Y 509.351,Z 500.473,A -85,B 0,C 180,E1 -5405.543,E2 -5405.543} C_VEL
LIN {X 0,Y 509.47,Z 495.249,A -85,B 0,C 180,E1 -5406.759,E2 -5406.759} C_VEL
LIN {X 0,Y 509.621,Z 488.911,A -85,B 0,C 180,E1 -5407.927,E2 -5407.927} C_VEL
LIN {X 0,Y 509.851,Z 480.841,A -85,B 0,C 180,E1 -5409.121,E2 -5409.121} C_VEL
LIN {X 0,Y 510.139,Z 472.576,A -85,B 0,C 180,E1 -5410.117,E2 -5410.117} C_VEL
LIN {X 0,Y 510.404,Z 462.427,A -85,B 0,C 180,E1 -5411.115,E2 -5411.115} C_VEL
LIN {X 0,Y 510.733,Z 450.695,A -85,B 0,C 180,E1 -5412.027,E2 -5412.027} C_VEL
LIN {X 0,Y 511.002,Z 439.542,A -85,B 0,C 180,E1 -5412.712,E2 -5412.712} C_VEL
LIN {X 0,Y 511.246,Z 427.882,A -85,B 0,C 180,E1 -5413.262,E2 -5413.262} C_VEL
LIN {X 0,Y 511.469,Z 414.493,A -85,B 0,C 180,E1 -5413.711,E2 -5413.711} C_VEL
LIN {X 0,Y 511.589,Z 401.419,A -85,B 0,C 180,E1 -5413.987,E2 -5413.987} C_VEL
LIN {X 0,Y 512.14,Z 310.199,A -85,B 0,C 180,E1 -5415.376,E2 -5415.376} C_VEL
LIN {X 0,Y 510.388,Z 301.417,A -85,B 0,C 180,E1 -5415.596,E2 -5415.596} C_VEL
LIN {X 0,Y 510.699,Z 288.09,A -85,B 0,C 180,E1 -5418.452,E2 -5418.452} C_VEL
LIN {X 0,Y 509.909,Z 281.972,A -85,B 0,C 180,E1 -5419.841,E2 -5419.841} C_VEL
LIN {X 0,Y 509.822,Z 281.981,A -85,B 0,C 180,E1 -5422.705,E2 -5422.705} C_VEL
LIN {X 0,Y 509.789,Z 281.988,A -85,B 0,C 180,E1 -5425.301,E2 -5425.301} C_VEL
LIN {X 0,Y 509.811,Z 281.979,A -85,B 0,C 180,E1 -5428.081,E2 -5428.081} C_VEL
LIN {X 0,Y 509.817,Z 281.982,A -85,B 0,C 180,E1 -5431.274,E2 -5431.274} C_VEL
LIN {X 0,Y 509.823,Z 281.979,A -85,B 0,C 180,E1 -5434.416,E2 -5434.416} C_VEL
LIN {X 0,Y 509.764,Z 281.986,A -85,B 0,C 180,E1 -5437.345,E2 -5437.345} C_VEL
LIN {X 0,Y 509.816,Z 281.98,A -85,B 0,C 180,E1 -5440.385,E2 -5440.385} C_VEL
LIN {X 0,Y 509.795,Z 281.98,A -85,B 0,C 180,E1 -5443.575,E2 -5443.575} C_VEL
LIN {X 0,Y 509.794,Z 281.986,A -85,B 0,C 180,E1 -5446.425,E2 -5446.425} C_VEL
LIN {X 0,Y 509.815,Z 281.978,A -85,B 0,C 180,E1 -5449.615,E2 -5449.615} C_VEL
LIN {X 0,Y 509.81,Z 281.982,A -85,B 0,C 180,E1 -5452.658,E2 -5452.658} C_VEL
LIN {X 0,Y 509.849,Z 281.977,A -85,B 0,C 180,E1 -5455.799,E2 -5455.799} C_VEL
LIN {X 0,Y 509.848,Z 281.978,A -85,B 0,C 180,E1 -5458.72,E2 -5458.72} C_VEL
LIN {X 0,Y 509.854,Z 281.978,A -85,B 0,C 180,E1 -5461.154,E2 -5461.154} C_VEL
LIN {X 0,Y 509.875,Z 281.976,A -85,B 0,C 180,E1 -5464.266,E2 -5464.266} C_VEL
LIN {X 0,Y 509.921,Z 282.194,A -85,B 0,C 180,E1 -5464.651,E2 -5464.651} C_VEL
LIN {X 0,Y 511.498,Z 290.457,A -85,B 0,C 180,E1 -5466.087,E2 -5466.087} C_VEL
LIN {X 0,Y 511.373,Z 299.727,A -85,B 0,C 180,E1 -5467.58,E2 -5467.58} C_VEL
LIN {X 0,Y 510.788,Z 318.473,A -85,B 0,C 180,E1 -5470.508,E2 -5470.508} C_VEL
LIN {X 0,Y 510.411,Z 334.644,A -85,B 0,C 180,E1 -5472.986,E2 -5472.986} C_VEL
LIN {X 0,Y 510.237,Z 344.145,A -85,B 0,C 180,E1 -5474.427,E2 -5474.427} C_VEL
LIN {X 0,Y 512.112,Z 358.344,A -85,B 0,C 180,E1 -5474.708,E2 -5474.708} C_VEL
LIN {X 0,Y 511.458,Z 453.801,A -85,B 0,C 180,E1 -5476.161,E2 -5476.161} C_VEL
LIN {X 0,Y 511.191,Z 467.501,A -85,B 0,C 180,E1 -5476.534,E2 -5476.534} C_VEL
LIN {X 0,Y 510.928,Z 479.937,A -85,B 0,C 180,E1 -5477.033,E2 -5477.033} C_VEL
LIN {X 0,Y 510.65,Z 492.186,A -85,B 0,C 180,E1 -5477.7,E2 -5477.7} C_VEL
LIN {X 0,Y 510.308,Z 503.434,A -85,B 0,C 180,E1 -5478.48,E2 -5478.48} C_VEL
LIN {X 0,Y 510.065,Z 513.827,A -85,B 0,C 180,E1 -5479.38,E2 -5479.38} C_VEL
LIN {X 0,Y 509.734,Z 523.977,A -85,B 0,C 180,E1 -5480.476,E2 -5480.476} C_VEL
LIN {X 0,Y 509.533,Z 532.924,A -85,B 0,C 180,E1 -5481.672,E2 -5481.672} C_VEL
LIN {X 0,Y 509.393,Z 540.04,A -85,B 0,C 180,E1 -5482.866,E2 -5482.866} C_VEL
LIN {X 0,Y 509.311,Z 545.727,A -85,B 0,C 180,E1 -5484.059,E2 -5484.059} C_VEL
LIN {X 0,Y 509.187,Z 550.188,A -85,B 0,C 180,E1 -5485.249,E2 -5485.249} C_VEL
LIN {X 0,Y 509.275,Z 552.559,A -85,B 0,C 180,E1 -5486.043,E2 -5486.043} C_VEL
LIN {X 0,Y 509.201,Z 554.48,A -85,B 0,C 180,E1 -5486.834,E2 -5486.834} C_VEL
LIN {X 0,Y 509.19,Z 555.917,A -85,B 0,C 180,E1 -5487.626,E2 -5487.626} C_VEL
LIN {X 0,Y 509.076,Z 557.57,A -85,B 0,C 180,E1 -5489.208,E2 -5489.208} C_VEL
LIN {X 0,Y 509.073,Z 557.802,A -85,B 0,C 180,E1 -5489.999,E2 -5489.999} C_VEL
LIN {X 0,Y 509.076,Z 557.588,A -85,B 0,C 180,E1 -5490.79,E2 -5490.79} C_VEL
LIN {X 0,Y 509.19,Z 555.973,A -85,B 0,C 180,E1 -5492.372,E2 -5492.372} C_VEL
LIN {X 0,Y 509.201,Z 554.551,A -85,B 0,C 180,E1 -5493.164,E2 -5493.164} C_VEL
LIN {X 0,Y 509.205,Z 551.57,A -85,B 0,C 180,E1 -5494.353,E2 -5494.353} C_VEL
LIN {X 0,Y 509.308,Z 547.531,A -85,B 0,C 180,E1 -5495.542,E2 -5495.542} C_VEL
LIN {X 0,Y 509.372,Z 541.749,A -85,B 0,C 180,E1 -5496.844,E2 -5496.844} C_VEL
LIN {X 0,Y 509.507,Z 534.48,A -85,B 0,C 180,E1 -5498.127,E2 -5498.127} C_VEL
LIN {X 0,Y 509.719,Z 526.015,A -85,B 0,C 180,E1 -5499.323,E2 -5499.323} C_VEL
LIN {X 0,Y 509.941,Z 517.284,A -85,B 0,C 180,E1 -5500.32,E2 -5500.32} C_VEL
LIN {X 0,Y 510.342,Z 506.539,A -85,B 0,C 180,E1 -5501.316,E2 -5501.316} C_VEL
LIN {X 0,Y 510.598,Z 495.12,A -85,B 0,C 180,E1 -5502.165,E2 -5502.165} C_VEL
LIN {X 0,Y 510.914,Z 483.954,A -85,B 0,C 180,E1 -5502.815,E2 -5502.815} C_VEL
LIN {X 0,Y 511.189,Z 471.61,A -85,B 0,C 180,E1 -5503.364,E2 -5503.364} C_VEL
LIN {X 0,Y 511.446,Z 459.03,A -85,B 0,C 180,E1 -5503.762,E2 -5503.762} C_VEL
LIN {X 0,Y 511.608,Z 444.538,A -85,B 0,C 180,E1 -5504.036,E2 -5504.036} C_VEL
LIN {X 0,Y 512.062,Z 357.027,A -85,B 0,C 180,E1 -5505.327,E2 -5505.327} C_VEL
LIN {X 0,Y 510.315,Z 344.983,A -85,B 0,C 180,E1 -5505.582,E2 -5505.582} C_VEL
LIN {X 0,Y 510.77,Z 325.001,A -85,B 0,C 180,E1 -5508.657,E2 -5508.657} C_VEL
LIN {X 0,Y 511.271,Z 307.569,A -85,B 0,C 180,E1 -5511.362,E2 -5511.362} C_VEL
LIN {X 0,Y 511.81,Z 292.871,A -85,B 0,C 180,E1 -5513.68,E2 -5513.68} C_VEL
LIN {X 0,Y 510.596,Z 285.354,A -85,B 0,C 180,E1 -5514.949,E2 -5514.949} C_VEL
LIN {X 0,Y 509.906,Z 281.972,A -85,B 0,C 180,E1 -5515.567,E2 -5515.567} C_VEL
LIN {X 0,Y 509.87,Z 281.971,A -85,B 0,C 180,E1 -5518.844,E2 -5518.844} C_VEL
LIN {X 0,Y 509.817,Z 281.978,A -85,B 0,C 180,E1 -5521.589,E2 -5521.589} C_VEL
LIN {X 0,Y 509.843,Z 281.975,A -85,B 0,C 180,E1 -5524.413,E2 -5524.413} C_VEL
LIN {X 0,Y 509.804,Z 281.979,A -85,B 0,C 180,E1 -5527.341,E2 -5527.341} C_VEL
LIN {X 0,Y 509.832,Z 281.975,A -85,B 0,C 180,E1 -5530.381,E2 -5530.381} C_VEL
LIN {X 0,Y 509.799,Z 281.979,A -85,B 0,C 180,E1 -5533.059,E2 -5533.059} C_VEL
LIN {X 0,Y 509.816,Z 281.982,A -85,B 0,C 180,E1 -5535.793,E2 -5535.793} C_VEL
LIN {X 0,Y 509.838,Z 281.974,A -85,B 0,C 180,E1 -5538.573,E2 -5538.573} C_VEL
LIN {X 0,Y 509.843,Z 281.977,A -85,B 0,C 180,E1 -5541.786,E2 -5541.786} C_VEL
LIN {X 0,Y 509.822,Z 281.976,A -85,B 0,C 180,E1 -5544.621,E2 -5544.621} C_VEL
LIN {X 0,Y 509.852,Z 281.979,A -85,B 0,C 180,E1 -5547.48,E2 -5547.48} C_VEL
LIN {X 0,Y 509.845,Z 281.973,A -85,B 0,C 180,E1 -5550.274,E2 -5550.274} C_VEL
LIN {X 0,Y 509.816,Z 281.98,A -85,B 0,C 180,E1 -5552.94,E2 -5552.94} C_VEL
LIN {X 0,Y 509.825,Z 281.978,A -85,B 0,C 180,E1 -5555.572,E2 -5555.572} C_VEL
LIN {X 0,Y 509.811,Z 281.978,A -85,B 0,C 180,E1 -5558.148,E2 -5558.148} C_VEL
LIN {X 0,Y 509.846,Z 281.977,A -85,B 0,C 180,E1 -5560.681,E2 -5560.681} C_VEL
LIN {X 0,Y 509.848,Z 281.978,A -85,B 0,C 180,E1 -5563.173,E2 -5563.173} C_VEL
LIN {X 0,Y 509.833,Z 281.975,A -85,B 0,C 180,E1 -5565.633,E2 -5565.633} C_VEL
LIN {X 0,Y 509.896,Z 281.973,A -85,B 0,C 180,E1 -5568.874,E2 -5568.874} C_VEL
LIN {X 0,Y 509.897,Z 281.969,A -85,B 0,C 180,E1 -5572.078,E2 -5572.078} C_VEL
LIN {X 0,Y 509.922,Z 281.968,A -85,B 0,C 180,E1 -5574.464,E2 -5574.464} C_VEL
LIN {X 0,Y 510.03,Z 281.951,A -85,B 0,C 180,E1 -5577.631,E2 -5577.631} C_VEL
LIN {X 0,Y 510.028,Z 281.955,A -85,B 0,C 180,E1 -5580.79,E2 -5580.79} C_VEL
LIN {X 0,Y 509.875,Z 281.971,A -85,B 0,C 180,E1 -5583.161,E2 -5583.161} C_VEL
LIN {X 0,Y 509.908,Z 281.97,A -85,B 0,C 180,E1 -5586.331,E2 -5586.331} C_VEL
LIN {X 0,Y 509.864,Z 281.973,A -85,B 0,C 180,E1 -5589.521,E2 -5589.521} C_VEL
LIN {X 0,Y 509.895,Z 281.971,A -85,B 0,C 180,E1 -5591.932,E2 -5591.932} C_VEL
LIN {X 0,Y 509.886,Z 281.969,A -85,B 0,C 180,E1 -5595.242,E2 -5595.242} C_VEL
LIN {X 0,Y 509.847,Z 281.976,A -85,B 0,C 180,E1 -5598.484,E2 -5598.484} C_VEL
LIN {X 0,Y 509.837,Z 281.975,A -85,B 0,C 180,E1 -5601.002,E2 -5601.002} C_VEL
LIN {X 0,Y 509.813,Z 281.982,A -85,B 0,C 180,E1 -5603.564,E2 -5603.564} C_VEL
LIN {X 0,Y 509.866,Z 281.973,A -85,B 0,C 180,E1 -5606.37,E2 -5606.37} C_VEL
LIN {X 0,Y 509.851,Z 281.977,A -85,B 0,C 180,E1 -5609.727,E2 -5609.727} C_VEL
LIN {X 0,Y 509.866,Z 281.972,A -85,B 0,C 180,E1 -5612.775,E2 -5612.775} C_VEL
LIN {X 0,Y 509.816,Z 281.981,A -85,B 0,C 180,E1 -5615.579,E2 -5615.579} C_VEL
LIN {X 0,Y 509.842,Z 281.975,A -85,B 0,C 180,E1 -5618.339,E2 -5618.339} C_VEL
LIN {X 0,Y 509.846,Z 281.978,A -85,B 0,C 180,E1 -5621.427,E2 -5621.427} C_VEL
LIN {X 0,Y 509.834,Z 281.977,A -85,B 0,C 180,E1 -5624.671,E2 -5624.671} C_VEL
LIN {X 0,Y 509.851,Z 281.973,A -85,B 0,C 180,E1 -5628.104,E2 -5628.104} C_VEL
LIN {X 0,Y 509.842,Z 281.977,A -85,B 0,C 180,E1 -5630.648,E2 -5630.648} C_VEL
LIN {X 0,Y 509.817,Z 281.979,A -85,B 0,C 180,E1 -5633.731,E2 -5633.731} C_VEL
LIN {X 0,Y 509.149,Z 282.063,A -85,B 0,C 180,E1 -5634.391,E2 -5634.391} C_VEL
LIN {X 0,Y 506.336,Z 282.414,A -85,B 0,C 180,E1 -5635.463,E2 -5635.463} C_VEL
LIN {X 0,Y 503.949,Z 282.713,A -85,B 0,C 180,E1 -5636.326,E2 -5636.326} C_VEL
LIN {X 0,Y 502.902,Z 282.843,A -85,B 0,C 180,E1 -5636.993,E2 -5636.993} C_VEL
LIN {X 0,Y 502.804,Z 282.853,A -85,B 0,C 180,E1 -5637.218,E2 -5637.218} C_VEL
LIN {X 0,Y 502.812,Z 282.85,A -85,B 0,C 180,E1 -5640.066,E2 -5640.066} C_VEL
LIN {X 0,Y 502.828,Z 282.853,A -85,B 0,C 180,E1 -5642.534,E2 -5642.534} C_VEL
LIN {X 0,Y 502.822,Z 282.851,A -85,B 0,C 180,E1 -5645.301,E2 -5645.301} C_VEL
LIN {X 0,Y 502.78,Z 282.854,A -85,B 0,C 180,E1 -5647.827,E2 -5647.827} C_VEL
LIN {X 0,Y 502.831,Z 282.853,A -85,B 0,C 180,E1 -5650.401,E2 -5650.401} C_VEL
LIN {X 0,Y 502.787,Z 282.862,A -85,B 0,C 180,E1 -5652.512,E2 -5652.512} C_VEL
LIN {X 0,Y 502.626,Z 283.053,A -85,B 0,C 180,E1 -5652.873,E2 -5652.873} C_VEL
LIN {X 0,Y 502.697,Z 292.776,A -85,B 0,C 180,E1 -5653.952,E2 -5653.952} C_VEL
LIN {X 0,Y 502.781,Z 295.04,A -85,B 0,C 180,E1 -5654.171,E2 -5654.171} C_VEL
LIN {X 0,Y 505.45,Z 312.261,A -85,B 0,C 180,E1 -5654.512,E2 -5654.512} C_VEL
LIN {X 0,Y 504.935,Z 406.571,A -85,B 0,C 180,E1 -5655.878,E2 -5655.878} C_VEL
LIN {X 0,Y 504.726,Z 420.245,A -85,B 0,C 180,E1 -5656.231,E2 -5656.231} C_VEL
LIN {X 0,Y 504.417,Z 432.39,A -85,B 0,C 180,E1 -5656.71,E2 -5656.71} C_VEL
LIN {X 0,Y 504.123,Z 444.987,A -85,B 0,C 180,E1 -5657.39,E2 -5657.39} C_VEL
LIN {X 0,Y 503.841,Z 455.616,A -85,B 0,C 180,E1 -5658.128,E2 -5658.128} C_VEL
LIN {X 0,Y 503.454,Z 466.064,A -85,B 0,C 180,E1 -5659.036,E2 -5659.036} C_VEL
LIN {X 0,Y 503.117,Z 476.336,A -85,B 0,C 180,E1 -5660.148,E2 -5660.148} C_VEL
LIN {X 0,Y 502.859,Z 483.916,A -85,B 0,C 180,E1 -5661.157,E2 -5661.157} C_VEL
LIN {X 0,Y 502.572,Z 491.318,A -85,B 0,C 180,E1 -5662.367,E2 -5662.367} C_VEL
LIN {X 0,Y 502.446,Z 497.259,A -85,B 0,C 180,E1 -5663.576,E2 -5663.576} C_VEL
LIN {X 0,Y 502.192,Z 501.966,A -85,B 0,C 180,E1 -5664.782,E2 -5664.782} C_VEL
LIN {X 0,Y 502.24,Z 505.556,A -85,B 0,C 180,E1 -5665.989,E2 -5665.989} C_VEL
LIN {X 0,Y 502.217,Z 507.407,A -85,B 0,C 180,E1 -5666.792,E2 -5666.792} C_VEL
LIN {X 0,Y 502.133,Z 508.829,A -85,B 0,C 180,E1 -5667.594,E2 -5667.594} C_VEL
LIN {X 0,Y 501.997,Z 510.441,A -85,B 0,C 180,E1 -5669.199,E2 -5669.199} C_VEL
LIN {X 0,Y 501.991,Z 510.678,A -85,B 0,C 180,E1 -5670.001,E2 -5670.001} C_VEL
LIN {X 0,Y 502.037,Z 509.912,A -85,B 0,C 180,E1 -5671.605,E2 -5671.605} C_VEL
LIN {X 0,Y 502.133,Z 508.95,A -85,B 0,C 180,E1 -5672.407,E2 -5672.407} C_VEL
LIN {X 0,Y 502.217,Z 507.595,A -85,B 0,C 180,E1 -5673.21,E2 -5673.21} C_VEL
LIN {X 0,Y 502.229,Z 504.749,A -85,B 0,C 180,E1 -5674.415,E2 -5674.415} C_VEL
LIN {X 0,Y 502.3,Z 500.877,A -85,B 0,C 180,E1 -5675.621,E2 -5675.621} C_VEL
LIN {X 0,Y 502.429,Z 495.867,A -85,B 0,C 180,E1 -5676.829,E2 -5676.829} C_VEL
LIN {X 0,Y 502.634,Z 489.543,A -85,B 0,C 180,E1 -5678.038,E2 -5678.038} C_VEL
LIN {X 0,Y 502.909,Z 481.677,A -85,B 0,C 180,E1 -5679.249,E2 -5679.249} C_VEL
LIN {X 0,Y 503.182,Z 473.638,A -85,B 0,C 180,E1 -5680.259,E2 -5680.259} C_VEL
LIN {X 0,Y 503.521,Z 463.785,A -85,B 0,C 180,E1 -5681.269,E2 -5681.269} C_VEL
LIN {X 0,Y 503.915,Z 452.079,A -85,B 0,C 180,E1 -5682.226,E2 -5682.226} C_VEL
LIN {X 0,Y 504.209,Z 441.893,A -85,B 0,C 180,E1 -5682.887,E2 -5682.887} C_VEL
LIN {X 0,Y 504.506,Z 429.801,A -85,B 0,C 180,E1 -5683.494,E2 -5683.494} C_VEL
LIN {X 0,Y 504.805,Z 416.485,A -85,B 0,C 180,E1 -5683.974,E2 -5683.974} C_VEL
LIN {X 0,Y 504.962,Z 403.025,A -85,B 0,C 180,E1 -5684.278,E2 -5684.278} C_VEL
LIN {X 0,Y 505.308,Z 310.977,A -85,B 0,C 180,E1 -5685.601,E2 -5685.601} C_VEL
LIN {X 0,Y 502.823,Z 295.032,A -85,B 0,C 180,E1 -5685.921,E2 -5685.921} C_VEL
LIN {X 0,Y 502.608,Z 285.975,A -85,B 0,C 180,E1 -5686.868,E2 -5686.868} C_VEL
LIN {X 0,Y 502.613,Z 282.883,A -85,B 0,C 180,E1 -5687.26,E2 -5687.26} C_VEL
LIN {X 0,Y 502.844,Z 282.848,A -85,B 0,C 180,E1 -5688.752,E2 -5688.752} C_VEL
LIN {X 0,Y 502.789,Z 282.858,A -85,B 0,C 180,E1 -5691.312,E2 -5691.312} C_VEL
LIN {X 0,Y 502.78,Z 282.856,A -85,B 0,C 180,E1 -5693.915,E2 -5693.915} C_VEL
LIN {X 0,Y 502.869,Z 282.843,A -85,B 0,C 180,E1 -5696.567,E2 -5696.567} C_VEL
LIN {X 0,Y 502.827,Z 282.853,A -85,B 0,C 180,E1 -5699.288,E2 -5699.288} C_VEL
LIN {X 0,Y 502.787,Z 282.853,A -85,B 0,C 180,E1 -5702.085,E2 -5702.085} C_VEL
LIN {X 0,Y 502.8,Z 282.854,A -85,B 0,C 180,E1 -5704.966,E2 -5704.966} C_VEL
LIN {X 0,Y 502.797,Z 282.852,A -85,B 0,C 180,E1 -5707.954,E2 -5707.954} C_VEL
LIN {X 0,Y 502.825,Z 282.853,A -85,B 0,C 180,E1 -5711.066,E2 -5711.066} C_VEL
LIN {X 0,Y 502.806,Z 282.852,A -85,B 0,C 180,E1 -5714.532,E2 -5714.532} C_VEL
LIN {X 0,Y 502.8,Z 282.851,A -85,B 0,C 180,E1 -5717.861,E2 -5717.861} C_VEL
LIN {X 0,Y 502.807,Z 282.857,A -85,B 0,C 180,E1 -5721.024,E2 -5721.024} C_VEL
LIN {X 0,Y 502.78,Z 282.853,A -85,B 0,C 180,E1 -5724.169,E2 -5724.169} C_VEL
LIN {X 0,Y 502.837,Z 282.852,A -85,B 0,C 180,E1 -5726.994,E2 -5726.994} C_VEL
LIN {X 0,Y 502.82,Z 282.848,A -85,B 0,C 180,E1 -5730.065,E2 -5730.065} C_VEL
LIN {X 0,Y 502.829,Z 282.851,A -85,B 0,C 180,E1 -5732.533,E2 -5732.533} C_VEL
LIN {X 0,Y 502.789,Z 282.852,A -85,B 0,C 180,E1 -5735.31,E2 -5735.31} C_VEL
LIN {X 0,Y 502.785,Z 282.852,A -85,B 0,C 180,E1 -5737.827,E2 -5737.827} C_VEL
LIN {X 0,Y 502.881,Z 282.873,A -85,B 0,C 180,E1 -5740.509,E2 -5740.509} C_VEL
LIN {X 0,Y 503.521,Z 288.742,A -85,B 0,C 180,E1 -5741.786,E2 -5741.786} C_VEL
LIN {X 0,Y 503.225,Z 300.613,A -85,B 0,C 180,E1 -5744.275,E2 -5744.275} C_VEL
LIN {X 0,Y 505.39,Z 312.477,A -85,B 0,C 180,E1 -5744.541,E2 -5744.541} C_VEL
LIN {X 0,Y 504.633,Z 408.229,A -85,B 0,C 180,E1 -5746.022,E2 -5746.022} C_VEL
LIN {X 0,Y 504.488,Z 421.703,A -85,B 0,C 180,E1 -5746.403,E2 -5746.403} C_VEL
LIN {X 0,Y 504.149,Z 433.948,A -85,B 0,C 180,E1 -5746.907,E2 -5746.907} C_VEL
LIN {X 0,Y 503.925,Z 445.574,A -85,B 0,C 180,E1 -5747.555,E2 -5747.555} C_VEL
LIN {X 0,Y 503.61,Z 457.783,A -85,B 0,C 180,E1 -5748.427,E2 -5748.427} C_VEL
LIN {X 0,Y 503.245,Z 467.883,A -85,B 0,C 180,E1 -5749.336,E2 -5749.336} C_VEL
LIN {X 0,Y 502.947,Z 476.999,A -85,B 0,C 180,E1 -5750.347,E2 -5750.347} C_VEL
LIN {X 0,Y 502.684,Z 485.883,A -85,B 0,C 180,E1 -5751.558,E2 -5751.558} C_VEL
LIN {X 0,Y 502.485,Z 492.985,A -85,B 0,C 180,E1 -5752.768,E2 -5752.768} C_VEL
LIN {X 0,Y 502.379,Z 498.641,A -85,B 0,C 180,E1 -5753.977,E2 -5753.977} C_VEL
LIN {X 0,Y 502.156,Z 503.091,A -85,B 0,C 180,E1 -5755.183,E2 -5755.183} C_VEL
LIN {X 0,Y 502.242,Z 505.43,A -85,B 0,C 180,E1 -5755.988,E2 -5755.988} C_VEL
LIN {X 0,Y 502.218,Z 507.348,A -85,B 0,C 180,E1 -5756.791,E2 -5756.791} C_VEL
LIN {X 0,Y 502.133,Z 508.811,A -85,B 0,C 180,E1 -5757.593,E2 -5757.593} C_VEL
LIN {X 0,Y 501.999,Z 510.496,A -85,B 0,C 180,E1 -5759.198,E2 -5759.198} C_VEL
LIN {X 0,Y 501.995,Z 510.754,A -85,B 0,C 180,E1 -5760,E2 -5760} C_VEL
LIN {X 0,Y 501.999,Z 510.577,A -85,B 0,C 180,E1 -5760.802,E2 -5760.802} C_VEL
LIN {X 0,Y 502.132,Z 509.018,A -85,B 0,C 180,E1 -5762.406,E2 -5762.406} C_VEL
LIN {X 0,Y 502.218,Z 507.64,A -85,B 0,C 180,E1 -5763.209,E2 -5763.209} C_VEL
LIN {X 0,Y 502.229,Z 504.729,A -85,B 0,C 180,E1 -5764.414,E2 -5764.414} C_VEL
LIN {X 0,Y 502.299,Z 500.764,A -85,B 0,C 180,E1 -5765.621,E2 -5765.621} C_VEL
LIN {X 0,Y 502.416,Z 495.082,A -85,B 0,C 180,E1 -5766.94,E2 -5766.94} C_VEL
LIN {X 0,Y 502.635,Z 487.904,A -85,B 0,C 180,E1 -5768.24,E2 -5768.24} C_VEL
LIN {X 0,Y 502.89,Z 479.523,A -85,B 0,C 180,E1 -5769.451,E2 -5769.451} C_VEL
LIN {X 0,Y 503.144,Z 470.848,A -85,B 0,C 180,E1 -5770.462,E2 -5770.462} C_VEL
LIN {X 0,Y 503.551,Z 460.138,A -85,B 0,C 180,E1 -5771.472,E2 -5771.472} C_VEL
LIN {X 0,Y 503.775,Z 449.925,A -85,B 0,C 180,E1 -5772.251,E2 -5772.251} C_VEL
LIN {X 0,Y 504.067,Z 439.455,A -85,B 0,C 180,E1 -5772.89,E2 -5772.89} C_VEL
LIN {X 0,Y 504.331,Z 427.612,A -85,B 0,C 180,E1 -5773.447,E2 -5773.447} C_VEL
LIN {X 0,Y 504.53,Z 414.009,A -85,B 0,C 180,E1 -5773.904,E2 -5773.904} C_VEL
LIN {X 0,Y 504.69,Z 400.272,A -85,B 0,C 180,E1 -5774.182,E2 -5774.182} C_VEL
LIN {X 0,Y 505.362,Z 311.349,A -85,B 0,C 180,E1 -5775.575,E2 -5775.575} C_VEL
LIN {X 0,Y 503.435,Z 301.94,A -85,B 0,C 180,E1 -5775.803,E2 -5775.803} C_VEL
LIN {X 0,Y 503.803,Z 289.772,A -85,B 0,C 180,E1 -5778.45,E2 -5778.45} C_VEL
LIN {X 0,Y 502.878,Z 282.846,A -85,B 0,C 180,E1 -5780.077,E2 -5780.077} C_VEL
LIN {X 0,Y 502.788,Z 282.859,A -85,B 0,C 180,E1 -5783.041,E2 -5783.041} C_VEL
LIN {X 0,Y 502.764,Z 282.86,A -85,B 0,C 180,E1 -5785.68,E2 -5785.68} C_VEL
LIN {X 0,Y 502.762,Z 282.858,A -85,B 0,C 180,E1 -5788.378,E2 -5788.378} C_VEL
LIN {X 0,Y 502.768,Z 282.858,A -85,B 0,C 180,E1 -5791.493,E2 -5791.493} C_VEL
LIN {X 0,Y 502.775,Z 282.857,A -85,B 0,C 180,E1 -5794.438,E2 -5794.438} C_VEL
LIN {X 0,Y 502.72,Z 282.865,A -85,B 0,C 180,E1 -5797.168,E2 -5797.168} C_VEL
LIN {X 0,Y 502.771,Z 282.855,A -85,B 0,C 180,E1 -5800.017,E2 -5800.017} C_VEL
LIN {X 0,Y 502.742,Z 282.86,A -85,B 0,C 180,E1 -5803.235,E2 -5803.235} C_VEL
LIN {X 0,Y 502.77,Z 282.855,A -85,B 0,C 180,E1 -5805.658,E2 -5805.658} C_VEL
LIN {X 0,Y 502.766,Z 282.857,A -85,B 0,C 180,E1 -5809.012,E2 -5809.012} C_VEL
LIN {X 0,Y 502.775,Z 282.859,A -85,B 0,C 180,E1 -5812.044,E2 -5812.044} C_VEL
LIN {X 0,Y 502.797,Z 282.853,A -85,B 0,C 180,E1 -5815.033,E2 -5815.033} C_VEL
LIN {X 0,Y 502.787,Z 282.86,A -85,B 0,C 180,E1 -5817.915,E2 -5817.915} C_VEL
LIN {X 0,Y 502.816,Z 282.856,A -85,B 0,C 180,E1 -5820.711,E2 -5820.711} C_VEL
LIN {X 0,Y 502.848,Z 282.851,A -85,B 0,C 180,E1 -5823.443,E2 -5823.443} C_VEL
LIN {X 0,Y 502.83,Z 282.854,A -85,B 0,C 180,E1 -5824.383,E2 -5824.383} C_VEL
LIN {X 0,Y 504.54,Z 291.638,A -85,B 0,C 180,E1 -5825.955,E2 -5825.955} C_VEL
LIN {X 0,Y 504.594,Z 296.86,A -85,B 0,C 180,E1 -5826.817,E2 -5826.817} C_VEL
LIN {X 0,Y 503.91,Z 316.869,A -85,B 0,C 180,E1 -5830.019,E2 -5830.019} C_VEL
LIN {X 0,Y 503.399,Z 335.62,A -85,B 0,C 180,E1 -5832.951,E2 -5832.951} C_VEL
LIN {X 0,Y 503.211,Z 343.741,A -85,B 0,C 180,E1 -5834.201,E2 -5834.201} C_VEL
LIN {X 0,Y 505.248,Z 359.142,A -85,B 0,C 180,E1 -5834.518,E2 -5834.518} C_VEL
LIN {X 0,Y 504.535,Z 453.495,A -85,B 0,C 180,E1 -5835.993,E2 -5835.993} C_VEL
LIN {X 0,Y 504.245,Z 467.142,A -85,B 0,C 180,E1 -5836.37,E2 -5836.37} C_VEL
LIN {X 0,Y 503.931,Z 480.068,A -85,B 0,C 180,E1 -5836.901,E2 -5836.901} C_VEL
LIN {X 0,Y 503.64,Z 492.43,A -85,B 0,C 180,E1 -5837.59,E2 -5837.59} C_VEL
LIN {X 0,Y 503.253,Z 504.058,A -85,B 0,C 180,E1 -5838.419,E2 -5838.419} C_VEL
LIN {X 0,Y 503.004,Z 514.224,A -85,B 0,C 180,E1 -5839.331,E2 -5839.331} C_VEL
LIN {X 0,Y 502.672,Z 523.437,A -85,B 0,C 180,E1 -5840.341,E2 -5840.341} C_VEL
LIN {X 0,Y 502.476,Z 532.435,A -85,B 0,C 180,E1 -5841.554,E2 -5841.554} C_VEL
LIN {X 0,Y 502.309,Z 539.596,A -85,B 0,C 180,E1 -5842.765,E2 -5842.765} C_VEL
LIN {X 0,Y 502.21,Z 545.314,A -85,B 0,C 180,E1 -5843.975,E2 -5843.975} C_VEL
LIN {X 0,Y 502.11,Z 549.804,A -85,B 0,C 180,E1 -5845.182,E2 -5845.182} C_VEL
LIN {X 0,Y 502.165,Z 552.189,A -85,B 0,C 180,E1 -5845.987,E2 -5845.987} C_VEL
LIN {X 0,Y 502.123,Z 554.123,A -85,B 0,C 180,E1 -5846.79,E2 -5846.79} C_VEL
LIN {X 0,Y 502.121,Z 555.572,A -85,B 0,C 180,E1 -5847.593,E2 -5847.593} C_VEL
LIN {X 0,Y 501.993,Z 557.238,A -85,B 0,C 180,E1 -5849.197,E2 -5849.197} C_VEL
LIN {X 0,Y 501.987,Z 557.473,A -85,B 0,C 180,E1 -5849.999,E2 -5849.999} C_VEL
LIN {X 0,Y 501.992,Z 557.26,A -85,B 0,C 180,E1 -5850.801,E2 -5850.801} C_VEL
LIN {X 0,Y 502.12,Z 555.643,A -85,B 0,C 180,E1 -5852.406,E2 -5852.406} C_VEL
LIN {X 0,Y 502.122,Z 554.214,A -85,B 0,C 180,E1 -5853.209,E2 -5853.209} C_VEL
LIN {X 0,Y 502.103,Z 551.221,A -85,B 0,C 180,E1 -5854.414,E2 -5854.414} C_VEL
LIN {X 0,Y 502.221,Z 547.167,A -85,B 0,C 180,E1 -5855.621,E2 -5855.621} C_VEL
LIN {X 0,Y 502.323,Z 541.008,A -85,B 0,C 180,E1 -5857.011,E2 -5857.011} C_VEL
LIN {X 0,Y 502.458,Z 534.067,A -85,B 0,C 180,E1 -5858.242,E2 -5858.242} C_VEL
LIN {X 0,Y 502.671,Z 525.565,A -85,B 0,C 180,E1 -5859.455,E2 -5859.455} C_VEL
LIN {X 0,Y 502.93,Z 516.797,A -85,B 0,C 180,E1 -5860.466,E2 -5860.466} C_VEL
LIN {X 0,Y 503.33,Z 506.008,A -85,B 0,C 180,E1 -5861.476,E2 -5861.476} C_VEL
LIN {X 0,Y 503.596,Z 495.602,A -85,B 0,C 180,E1 -5862.264,E2 -5862.264} C_VEL
LIN {X 0,Y 503.938,Z 483.269,A -85,B 0,C 180,E1 -5862.995,E2 -5862.995} C_VEL
LIN {X 0,Y 504.272,Z 470.83,A -85,B 0,C 180,E1 -5863.55,E2 -5863.55} C_VEL
LIN {X 0,Y 504.537,Z 458.026,A -85,B 0,C 180,E1 -5863.954,E2 -5863.954} C_VEL
LIN {X 0,Y 504.72,Z 443.086,A -85,B 0,C 180,E1 -5864.231,E2 -5864.231} C_VEL
LIN {X 0,Y 505.137,Z 357.396,A -85,B 0,C 180,E1 -5865.532,E2 -5865.532} C_VEL
LIN {X 0,Y 503.301,Z 344.707,A -85,B 0,C 180,E1 -5865.805,E2 -5865.805} C_VEL
LIN {X 0,Y 503.775,Z 326.055,A -85,B 0,C 180,E1 -5868.714,E2 -5868.714} C_VEL
LIN {X 0,Y 504.407,Z 307.336,A -85,B 0,C 180,E1 -5871.667,E2 -5871.667} C_VEL
LIN {X 0,Y 504.873,Z 293.969,A -85,B 0,C 180,E1 -5873.808,E2 -5873.808} C_VEL
LIN {X 0,Y 503.199,Z 284.437,A -85,B 0,C 180,E1 -5875.45,E2 -5875.45} C_VEL
LIN {X 0,Y 502.869,Z 282.849,A -85,B 0,C 180,E1 -5875.756,E2 -5875.756} C_VEL
LIN {X 0,Y 502.835,Z 282.852,A -85,B 0,C 180,E1 -5878.372,E2 -5878.372} C_VEL
LIN {X 0,Y 502.79,Z 282.853,A -85,B 0,C 180,E1 -5881.498,E2 -5881.498} C_VEL
LIN {X 0,Y 502.801,Z 282.858,A -85,B 0,C 180,E1 -5883.993,E2 -5883.993} C_VEL
LIN {X 0,Y 502.761,Z 282.856,A -85,B 0,C 180,E1 -5887.175,E2 -5887.175} C_VEL
LIN {X 0,Y 502.783,Z 282.857,A -85,B 0,C 180,E1 -5890.014,E2 -5890.014} C_VEL
LIN {X 0,Y 502.798,Z 282.853,A -85,B 0,C 180,E1 -5892.198,E2 -5892.198} C_VEL
LIN {X 0,Y 502.78,Z 282.858,A -85,B 0,C 180,E1 -5895.469,E2 -5895.469} C_VEL
LIN {X 0,Y 502.789,Z 282.856,A -85,B 0,C 180,E1 -5897.86,E2 -5897.86} C_VEL
LIN {X 0,Y 502.786,Z 282.854,A -85,B 0,C 180,E1 -5901.022,E2 -5901.022} C_VEL
LIN {X 0,Y 502.767,Z 282.855,A -85,B 0,C 180,E1 -5904.168,E2 -5904.168} C_VEL
LIN {X 0,Y 502.823,Z 282.851,A -85,B 0,C 180,E1 -5906.993,E2 -5906.993} C_VEL
LIN {X 0,Y 502.802,Z 282.851,A -85,B 0,C 180,E1 -5910.065,E2 -5910.065} C_VEL
LIN {X 0,Y 502.775,Z 282.859,A -85,B 0,C 180,E1 -5913.429,E2 -5913.429} C_VEL
LIN {X 0,Y 502.756,Z 282.857,A -85,B 0,C 180,E1 -5916.084,E2 -5916.084} C_VEL
LIN {X 0,Y 502.771,Z 282.857,A -85,B 0,C 180,E1 -5918.688,E2 -5918.688} C_VEL
LIN {X 0,Y 502.812,Z 282.854,A -85,B 0,C 180,E1 -5921.248,E2 -5921.248} C_VEL
LIN {X 0,Y 502.828,Z 282.851,A -85,B 0,C 180,E1 -5924.663,E2 -5924.663} C_VEL
LIN {X 0,Y 502.867,Z 282.844,A -85,B 0,C 180,E1 -5928.039,E2 -5928.039} C_VEL
LIN {X 0,Y 502.847,Z 282.848,A -85,B 0,C 180,E1 -5931.156,E2 -5931.156} C_VEL
LIN {X 0,Y 502.838,Z 282.847,A -85,B 0,C 180,E1 -5933.58,E2 -5933.58} C_VEL
LIN {X 0,Y 502.85,Z 282.851,A -85,B 0,C 180,E1 -5936.795,E2 -5936.795} C_VEL
LIN {X 0,Y 502.888,Z 282.844,A -85,B 0,C 180,E1 -5938.398,E2 -5938.398} C_VEL
LIN {X 0,Y 502.979,Z 282.833,A -85,B 0,C 180,E1 -5940.801,E2 -5940.801} C_VEL
LIN {X 0,Y 502.995,Z 282.831,A -85,B 0,C 180,E1 -5942.402,E2 -5942.402} C_VEL
LIN {X 0,Y 502.885,Z 282.842,A -85,B 0,C 180,E1 -5945.614,E2 -5945.614} C_VEL
LIN {X 0,Y 502.838,Z 282.85,A -85,B 0,C 180,E1 -5948.034,E2 -5948.034} C_VEL
LIN {X 0,Y 502.865,Z 282.844,A -85,B 0,C 180,E1 -5951.284,E2 -5951.284} C_VEL
LIN {X 0,Y 502.823,Z 282.852,A -85,B 0,C 180,E1 -5954.572,E2 -5954.572} C_VEL
LIN {X 0,Y 502.808,Z 282.854,A -85,B 0,C 180,E1 -5957.909,E2 -5957.909} C_VEL
LIN {X 0,Y 502.821,Z 282.851,A -85,B 0,C 180,E1 -5960.537,E2 -5960.537} C_VEL
LIN {X 0,Y 502.78,Z 282.855,A -85,B 0,C 180,E1 -5963.041,E2 -5963.041} C_VEL
LIN {X 0,Y 502.785,Z 282.857,A -85,B 0,C 180,E1 -5965.679,E2 -5965.679} C_VEL
LIN {X 0,Y 502.788,Z 282.855,A -85,B 0,C 180,E1 -5968.376,E2 -5968.376} C_VEL
LIN {X 0,Y 502.787,Z 282.856,A -85,B 0,C 180,E1 -5971.144,E2 -5971.144} C_VEL
LIN {X 0,Y 502.796,Z 282.856,A -85,B 0,C 180,E1 -5973.995,E2 -5973.995} C_VEL
LIN {X 0,Y 502.758,Z 282.861,A -85,B 0,C 180,E1 -5977.177,E2 -5977.177} C_VEL
LIN {X 0,Y 502.781,Z 282.856,A -85,B 0,C 180,E1 -5980.016,E2 -5980.016} C_VEL
LIN {X 0,Y 502.798,Z 282.853,A -85,B 0,C 180,E1 -5982.2,E2 -5982.2} C_VEL
LIN {X 0,Y 502.781,Z 282.858,A -85,B 0,C 180,E1 -5985.471,E2 -5985.471} C_VEL
LIN {X 0,Y 502.815,Z 282.855,A -85,B 0,C 180,E1 -5988.935,E2 -5988.935} C_VEL
LIN {X 0,Y 502.789,Z 282.853,A -85,B 0,C 180,E1 -5992.047,E2 -5992.047} C_VEL
LIN {X 0,Y 502.792,Z 282.856,A -85,B 0,C 180,E1 -5995.035,E2 -5995.035} C_VEL
LIN {X 0,Y 502.804,Z 282.853,A -85,B 0,C 180,E1 -5997.218,E2 -5997.218} C_VEL
LIN {X 0,Y 502.103,Z 282.939,A -85,B 0,C 180,E1 -5997.887,E2 -5997.887} C_VEL
LIN {X 0,Y 499.239,Z 283.299,A -85,B 0,C 180,E1 -5998.973,E2 -5998.973} C_VEL
LIN {X 0,Y 496.845,Z 283.595,A -85,B 0,C 180,E1 -5999.848,E2 -5999.848} C_VEL
LIN {X 0,Y 495.828,Z 283.724,A -85,B 0,C 180,E1 -6000.523,E2 -6000.523} C_VEL
LIN {X 0,Y 495.749,Z 283.73,A -85,B 0,C 180,E1 -6000.752,E2 -6000.752} C_VEL
LIN {X 0,Y 495.789,Z 283.725,A -85,B 0,C 180,E1 -6003.933,E2 -6003.933} C_VEL
LIN {X 0,Y 495.759,Z 283.732,A -85,B 0,C 180,E1 -6007.141,E2 -6007.141} C_VEL
LIN {X 0,Y 495.775,Z 283.729,A -85,B 0,C 180,E1 -6010.111,E2 -6010.111} C_VEL
LIN {X 0,Y 495.854,Z 283.721,A -85,B 0,C 180,E1 -6011.832,E2 -6011.832} C_VEL
LIN {X 0,Y 495.58,Z 283.956,A -85,B 0,C 180,E1 -6012.834,E2 -6012.834} C_VEL
LIN {X 0,Y 495.744,Z 292.757,A -85,B 0,C 180,E1 -6013.741,E2 -6013.741} C_VEL
LIN {X 0,Y 495.886,Z 295.437,A -85,B 0,C 180,E1 -6013.951,E2 -6013.951} C_VEL
LIN {X 0,Y 498.638,Z 313.464,A -85,B 0,C 180,E1 -6014.309,E2 -6014.309} C_VEL
LIN {X 0,Y 498.038,Z 408.053,A -85,B 0,C 180,E1 -6015.704,E2 -6015.704} C_VEL
LIN {X 0,Y 497.85,Z 421.273,A -85,B 0,C 180,E1 -6016.063,E2 -6016.063} C_VEL
LIN {X 0,Y 497.515,Z 433.728,A -85,B 0,C 180,E1 -6016.574,E2 -6016.574} C_VEL
LIN {X 0,Y 497.194,Z 445.91,A -85,B 0,C 180,E1 -6017.25,E2 -6017.25} C_VEL
LIN {X 0,Y 496.866,Z 457.172,A -85,B 0,C 180,E1 -6018.062,E2 -6018.062} C_VEL
LIN {X 0,Y 496.418,Z 468.427,A -85,B 0,C 180,E1 -6019.086,E2 -6019.086} C_VEL
LIN {X 0,Y 496.107,Z 476.645,A -85,B 0,C 180,E1 -6020.007,E2 -6020.007} C_VEL
LIN {X 0,Y 495.835,Z 484.228,A -85,B 0,C 180,E1 -6021.031,E2 -6021.031} C_VEL
LIN {X 0,Y 495.519,Z 491.632,A -85,B 0,C 180,E1 -6022.257,E2 -6022.257} C_VEL
LIN {X 0,Y 495.368,Z 497.575,A -85,B 0,C 180,E1 -6023.484,E2 -6023.484} C_VEL
LIN {X 0,Y 495.134,Z 502.281,A -85,B 0,C 180,E1 -6024.707,E2 -6024.707} C_VEL
LIN {X 0,Y 495.176,Z 505.872,A -85,B 0,C 180,E1 -6025.931,E2 -6025.931} C_VEL
LIN {X 0,Y 495.134,Z 507.724,A -85,B 0,C 180,E1 -6026.746,E2 -6026.746} C_VEL
LIN {X 0,Y 495.069,Z 509.145,A -85,B 0,C 180,E1 -6027.56,E2 -6027.56} C_VEL
LIN {X 0,Y 494.917,Z 510.757,A -85,B 0,C 180,E1 -6029.187,E2 -6029.187} C_VEL
LIN {X 0,Y 494.908,Z 510.994,A -85,B 0,C 180,E1 -6030.001,E2 -6030.001} C_VEL
LIN {X 0,Y 494.964,Z 510.227,A -85,B 0,C 180,E1 -6031.628,E2 -6031.628} C_VEL
LIN {X 0,Y 495.069,Z 509.264,A -85,B 0,C 180,E1 -6032.442,E2 -6032.442} C_VEL
LIN {X 0,Y 495.134,Z 507.91,A -85,B 0,C 180,E1 -6033.256,E2 -6033.256} C_VEL
LIN {X 0,Y 495.158,Z 505.062,A -85,B 0,C 180,E1 -6034.478,E2 -6034.478} C_VEL
LIN {X 0,Y 495.251,Z 501.188,A -85,B 0,C 180,E1 -6035.702,E2 -6035.702} C_VEL
LIN {X 0,Y 495.374,Z 496.176,A -85,B 0,C 180,E1 -6036.927,E2 -6036.927} C_VEL
LIN {X 0,Y 495.598,Z 489.849,A -85,B 0,C 180,E1 -6038.153,E2 -6038.153} C_VEL
LIN {X 0,Y 495.885,Z 481.979,A -85,B 0,C 180,E1 -6039.381,E2 -6039.381} C_VEL
LIN {X 0,Y 496.198,Z 473.935,A -85,B 0,C 180,E1 -6040.405,E2 -6040.405} C_VEL
LIN {X 0,Y 496.577,Z 464.074,A -85,B 0,C 180,E1 -6041.429,E2 -6041.429} C_VEL
LIN {X 0,Y 496.983,Z 452.59,A -85,B 0,C 180,E1 -6042.382,E2 -6042.382} C_VEL
LIN {X 0,Y 497.303,Z 442.163,A -85,B 0,C 180,E1 -6043.069,E2 -6043.069} C_VEL
LIN {X 0,Y 497.61,Z 430.049,A -85,B 0,C 180,E1 -6043.685,E2 -6043.685} C_VEL
LIN {X 0,Y 497.918,Z 416.701,A -85,B 0,C 180,E1 -6044.171,E2 -6044.171} C_VEL
LIN {X 0,Y 498.091,Z 403.138,A -85,B 0,C 180,E1 -6044.479,E2 -6044.479} C_VEL
LIN {X 0,Y 498.533,Z 312.07,A -85,B 0,C 180,E1 -6045.805,E2 -6045.805} C_VEL
LIN {X 0,Y 495.816,Z 294.868,A -85,B 0,C 180,E1 -6046.16,E2 -6046.16} C_VEL
LIN {X 0,Y 495.589,Z 285.203,A -85,B 0,C 180,E1 -6047.114,E2 -6047.114} C_VEL
LIN {X 0,Y 495.591,Z 283.758,A -85,B 0,C 180,E1 -6047.3,E2 -6047.3} C_VEL
LIN {X 0,Y 495.837,Z 283.723,A -85,B 0,C 180,E1 -6048.257,E2 -6048.257} C_VEL
LIN {X 0,Y 495.779,Z 283.727,A -85,B 0,C 180,E1 -6050.757,E2 -6050.757} C_VEL
LIN {X 0,Y 495.748,Z 283.734,A -85,B 0,C 180,E1 -6053.388,E2 -6053.388} C_VEL
LIN {X 0,Y 495.828,Z 283.721,A -85,B 0,C 180,E1 -6056.75,E2 -6056.75} C_VEL
LIN {X 0,Y 495.77,Z 283.73,A -85,B 0,C 180,E1 -6059.747,E2 -6059.747} C_VEL
LIN {X 0,Y 495.771,Z 283.728,A -85,B 0,C 180,E1 -6062.595,E2 -6062.595} C_VEL
LIN {X 0,Y 495.752,Z 283.733,A -85,B 0,C 180,E1 -6065.538,E2 -6065.538} C_VEL
LIN {X 0,Y 495.768,Z 283.729,A -85,B 0,C 180,E1 -6068.768,E2 -6068.768} C_VEL
LIN {X 0,Y 495.761,Z 283.729,A -85,B 0,C 180,E1 -6071.781,E2 -6071.781} C_VEL
LIN {X 0,Y 495.755,Z 283.736,A -85,B 0,C 180,E1 -6075.14,E2 -6075.14} C_VEL
LIN {X 0,Y 495.761,Z 283.728,A -85,B 0,C 180,E1 -6078.219,E2 -6078.219} C_VEL
LIN {X 0,Y 495.756,Z 283.73,A -85,B 0,C 180,E1 -6081.409,E2 -6081.409} C_VEL
LIN {X 0,Y 495.753,Z 283.73,A -85,B 0,C 180,E1 -6084.462,E2 -6084.462} C_VEL
LIN {X 0,Y 495.772,Z 283.727,A -85,B 0,C 180,E1 -6087.406,E2 -6087.406} C_VEL
LIN {X 0,Y 495.771,Z 283.727,A -85,B 0,C 180,E1 -6090.254,E2 -6090.254} C_VEL
LIN {X 0,Y 495.811,Z 283.722,A -85,B 0,C 180,E1 -6093.255,E2 -6093.255} C_VEL
LIN {X 0,Y 495.748,Z 283.735,A -85,B 0,C 180,E1 -6096.613,E2 -6096.613} C_VEL
LIN {X 0,Y 495.784,Z 283.728,A -85,B 0,C 180,E1 -6099.324,E2 -6099.324} C_VEL
LIN {X 0,Y 495.834,Z 283.802,A -85,B 0,C 180,E1 -6100.382,E2 -6100.382} C_VEL
LIN {X 0,Y 496.527,Z 290.521,A -85,B 0,C 180,E1 -6101.857,E2 -6101.857} C_VEL
LIN {X 0,Y 496.273,Z 300.894,A -85,B 0,C 180,E1 -6104.056,E2 -6104.056} C_VEL
LIN {X 0,Y 498.555,Z 312.555,A -85,B 0,C 180,E1 -6104.325,E2 -6104.325} C_VEL
LIN {X 0,Y 497.753,Z 407.698,A -85,B 0,C 180,E1 -6105.825,E2 -6105.825} C_VEL
LIN {X 0,Y 497.576,Z 421.41,A -85,B 0,C 180,E1 -6106.211,E2 -6106.211} C_VEL
LIN {X 0,Y 497.208,Z 433.825,A -85,B 0,C 180,E1 -6106.721,E2 -6106.721} C_VEL
LIN {X 0,Y 496.959,Z 446.242,A -85,B 0,C 180,E1 -6107.423,E2 -6107.423} C_VEL
LIN {X 0,Y 496.652,Z 457.823,A -85,B 0,C 180,E1 -6108.263,E2 -6108.263} C_VEL
LIN {X 0,Y 496.279,Z 467.993,A -85,B 0,C 180,E1 -6109.185,E2 -6109.185} C_VEL
LIN {X 0,Y 495.939,Z 477.151,A -85,B 0,C 180,E1 -6110.209,E2 -6110.209} C_VEL
LIN {X 0,Y 495.642,Z 486.074,A -85,B 0,C 180,E1 -6111.438,E2 -6111.438} C_VEL
LIN {X 0,Y 495.429,Z 493.217,A -85,B 0,C 180,E1 -6112.665,E2 -6112.665} C_VEL
LIN {X 0,Y 495.318,Z 498.898,A -85,B 0,C 180,E1 -6113.891,E2 -6113.891} C_VEL
LIN {X 0,Y 495.077,Z 503.371,A -85,B 0,C 180,E1 -6115.114,E2 -6115.114} C_VEL
LIN {X 0,Y 495.178,Z 505.724,A -85,B 0,C 180,E1 -6115.931,E2 -6115.931} C_VEL
LIN {X 0,Y 495.135,Z 507.652,A -85,B 0,C 180,E1 -6116.745,E2 -6116.745} C_VEL
LIN {X 0,Y 495.069,Z 509.125,A -85,B 0,C 180,E1 -6117.559,E2 -6117.559} C_VEL
LIN {X 0,Y 494.919,Z 510.824,A -85,B 0,C 180,E1 -6119.186,E2 -6119.186} C_VEL
LIN {X 0,Y 494.912,Z 511.085,A -85,B 0,C 180,E1 -6120,E2 -6120} C_VEL
LIN {X 0,Y 494.919,Z 510.908,A -85,B 0,C 180,E1 -6120.814,E2 -6120.814} C_VEL
LIN {X 0,Y 495.068,Z 509.344,A -85,B 0,C 180,E1 -6122.441,E2 -6122.441} C_VEL
LIN {X 0,Y 495.135,Z 507.961,A -85,B 0,C 180,E1 -6123.255,E2 -6123.255} C_VEL
LIN {X 0,Y 495.158,Z 505.038,A -85,B 0,C 180,E1 -6124.477,E2 -6124.477} C_VEL
LIN {X 0,Y 495.25,Z 501.054,A -85,B 0,C 180,E1 -6125.701,E2 -6125.701} C_VEL
LIN {X 0,Y 495.38,Z 494.992,A -85,B 0,C 180,E1 -6127.11,E2 -6127.11} C_VEL
LIN {X 0,Y 495.598,Z 488.14,A -85,B 0,C 180,E1 -6128.358,E2 -6128.358} C_VEL
LIN {X 0,Y 495.882,Z 479.716,A -85,B 0,C 180,E1 -6129.586,E2 -6129.586} C_VEL
LIN {X 0,Y 496.139,Z 470.998,A -85,B 0,C 180,E1 -6130.612,E2 -6130.612} C_VEL
LIN {X 0,Y 496.593,Z 460.235,A -85,B 0,C 180,E1 -6131.635,E2 -6131.635} C_VEL
LIN {X 0,Y 496.846,Z 449.179,A -85,B 0,C 180,E1 -6132.478,E2 -6132.478} C_VEL
LIN {X 0,Y 497.145,Z 437.417,A -85,B 0,C 180,E1 -6133.177,E2 -6133.177} C_VEL
LIN {X 0,Y 497.451,Z 424.86,A -85,B 0,C 180,E1 -6133.741,E2 -6133.741} C_VEL
LIN {X 0,Y 497.653,Z 412.699,A -85,B 0,C 180,E1 -6134.126,E2 -6134.126} C_VEL
LIN {X 0,Y 497.803,Z 396.129,A -85,B 0,C 180,E1 -6134.434,E2 -6134.434} C_VEL
LIN {X 0,Y 498.495,Z 312.076,A -85,B 0,C 180,E1 -6135.797,E2 -6135.797} C_VEL
LIN {X 0,Y 496.509,Z 302.416,A -85,B 0,C 180,E1 -6136.039,E2 -6136.039} C_VEL
LIN {X 0,Y 496.837,Z 290.839,A -85,B 0,C 180,E1 -6138.603,E2 -6138.603} C_VEL
LIN {X 0,Y 495.813,Z 283.726,A -85,B 0,C 180,E1 -6140.314,E2 -6140.314} C_VEL
LIN {X 0,Y 495.738,Z 283.738,A -85,B 0,C 180,E1 -6143.388,E2 -6143.388} C_VEL
LIN {X 0,Y 495.71,Z 283.737,A -85,B 0,C 180,E1 -6146.073,E2 -6146.073} C_VEL
LIN {X 0,Y 495.698,Z 283.741,A -85,B 0,C 180,E1 -6148.82,E2 -6148.82} C_VEL
LIN {X 0,Y 495.732,Z 283.733,A -85,B 0,C 180,E1 -6151.72,E2 -6151.72} C_VEL
LIN {X 0,Y 495.745,Z 283.735,A -85,B 0,C 180,E1 -6154.689,E2 -6154.689} C_VEL
LIN {X 0,Y 495.694,Z 283.738,A -85,B 0,C 180,E1 -6157.565,E2 -6157.565} C_VEL
LIN {X 0,Y 495.744,Z 283.73,A -85,B 0,C 180,E1 -6160.044,E2 -6160.044} C_VEL
LIN {X 0,Y 495.694,Z 283.741,A -85,B 0,C 180,E1 -6162.887,E2 -6162.887} C_VEL
LIN {X 0,Y 495.716,Z 283.736,A -85,B 0,C 180,E1 -6165.996,E2 -6165.996} C_VEL
LIN {X 0,Y 495.729,Z 283.733,A -85,B 0,C 180,E1 -6169.296,E2 -6169.296} C_VEL
LIN {X 0,Y 495.731,Z 283.732,A -85,B 0,C 180,E1 -6171.406,E2 -6171.406} C_VEL
LIN {X 0,Y 495.747,Z 283.735,A -85,B 0,C 180,E1 -6174.461,E2 -6174.461} C_VEL
LIN {X 0,Y 495.771,Z 283.73,A -85,B 0,C 180,E1 -6177.405,E2 -6177.405} C_VEL
LIN {X 0,Y 495.766,Z 283.738,A -85,B 0,C 180,E1 -6180.253,E2 -6180.253} C_VEL
LIN {X 0,Y 495.778,Z 283.731,A -85,B 0,C 180,E1 -6183.262,E2 -6183.262} C_VEL
LIN {X 0,Y 495.823,Z 283.857,A -85,B 0,C 180,E1 -6184.159,E2 -6184.159} C_VEL
LIN {X 0,Y 497.606,Z 292.926,A -85,B 0,C 180,E1 -6185.821,E2 -6185.821} C_VEL
LIN {X 0,Y 497.686,Z 298.14,A -85,B 0,C 180,E1 -6186.708,E2 -6186.708} C_VEL
LIN {X 0,Y 496.95,Z 317.961,A -85,B 0,C 180,E1 -6189.943,E2 -6189.943} C_VEL
LIN {X 0,Y 496.374,Z 336.67,A -85,B 0,C 180,E1 -6192.914,E2 -6192.914} C_VEL
LIN {X 0,Y 496.179,Z 343.277,A -85,B 0,C 180,E1 -6193.952,E2 -6193.952} C_VEL
LIN {X 0,Y 498.404,Z 359.92,A -85,B 0,C 180,E1 -6194.314,E2 -6194.314} C_VEL
LIN {X 0,Y 497.619,Z 453.273,A -85,B 0,C 180,E1 -6195.82,E2 -6195.82} C_VEL
LIN {X 0,Y 497.303,Z 466.836,A -85,B 0,C 180,E1 -6196.202,E2 -6196.202} C_VEL
LIN {X 0,Y 496.976,Z 479.223,A -85,B 0,C 180,E1 -6196.714,E2 -6196.714} C_VEL
LIN {X 0,Y 496.682,Z 491.032,A -85,B 0,C 180,E1 -6197.371,E2 -6197.371} C_VEL
LIN {X 0,Y 496.262,Z 503.39,A -85,B 0,C 180,E1 -6198.253,E2 -6198.253} C_VEL
LIN {X 0,Y 495.929,Z 513.632,A -85,B 0,C 180,E1 -6199.177,E2 -6199.177} C_VEL
LIN {X 0,Y 495.619,Z 522.898,A -85,B 0,C 180,E1 -6200.202,E2 -6200.202} C_VEL
LIN {X 0,Y 495.418,Z 531.944,A -85,B 0,C 180,E1 -6201.433,E2 -6201.433} C_VEL
LIN {X 0,Y 495.249,Z 539.154,A -85,B 0,C 180,E1 -6202.662,E2 -6202.662} C_VEL
LIN {X 0,Y 495.111,Z 545.484,A -85,B 0,C 180,E1 -6204.029,E2 -6204.029} C_VEL
LIN {X 0,Y 495.037,Z 549.425,A -85,B 0,C 180,E1 -6205.113,E2 -6205.113} C_VEL
LIN {X 0,Y 495.056,Z 551.819,A -85,B 0,C 180,E1 -6205.929,E2 -6205.929} C_VEL
LIN {X 0,Y 495.045,Z 553.766,A -85,B 0,C 180,E1 -6206.744,E2 -6206.744} C_VEL
LIN {X 0,Y 495.025,Z 555.225,A -85,B 0,C 180,E1 -6207.558,E2 -6207.558} C_VEL
LIN {X 0,Y 494.963,Z 556.265,A -85,B 0,C 180,E1 -6208.372,E2 -6208.372} C_VEL
LIN {X 0,Y 494.913,Z 556.907,A -85,B 0,C 180,E1 -6209.186,E2 -6209.186} C_VEL
LIN {X 0,Y 494.905,Z 557.145,A -85,B 0,C 180,E1 -6209.999,E2 -6209.999} C_VEL
LIN {X 0,Y 494.912,Z 556.933,A -85,B 0,C 180,E1 -6210.813,E2 -6210.813} C_VEL
LIN {X 0,Y 494.963,Z 556.321,A -85,B 0,C 180,E1 -6211.626,E2 -6211.626} C_VEL
LIN {X 0,Y 495.024,Z 555.311,A -85,B 0,C 180,E1 -6212.44,E2 -6212.44} C_VEL
LIN {X 0,Y 495.045,Z 553.877,A -85,B 0,C 180,E1 -6213.255,E2 -6213.255} C_VEL
LIN {X 0,Y 495.008,Z 550.873,A -85,B 0,C 180,E1 -6214.478,E2 -6214.478} C_VEL
LIN {X 0,Y 495.134,Z 546.803,A -85,B 0,C 180,E1 -6215.701,E2 -6215.701} C_VEL
LIN {X 0,Y 495.252,Z 540.515,A -85,B 0,C 180,E1 -6217.132,E2 -6217.132} C_VEL
LIN {X 0,Y 495.381,Z 533.652,A -85,B 0,C 180,E1 -6218.361,E2 -6218.361} C_VEL
LIN {X 0,Y 495.601,Z 525.11,A -85,B 0,C 180,E1 -6219.591,E2 -6219.591} C_VEL
LIN {X 0,Y 495.896,Z 516.306,A -85,B 0,C 180,E1 -6220.616,E2 -6220.616} C_VEL
LIN {X 0,Y 496.309,Z 505.475,A -85,B 0,C 180,E1 -6221.641,E2 -6221.641} C_VEL
LIN {X 0,Y 496.634,Z 494.679,A -85,B 0,C 180,E1 -6222.462,E2 -6222.462} C_VEL
LIN {X 0,Y 496.96,Z 482.587,A -85,B 0,C 180,E1 -6223.181,E2 -6223.181} C_VEL
LIN {X 0,Y 497.353,Z 470.05,A -85,B 0,C 180,E1 -6223.742,E2 -6223.742} C_VEL
LIN {X 0,Y 497.62,Z 458.011,A -85,B 0,C 180,E1 -6224.126,E2 -6224.126} C_VEL
LIN {X 0,Y 497.805,Z 443.304,A -85,B 0,C 180,E1 -6224.407,E2 -6224.407} C_VEL
LIN {X 0,Y 498.323,Z 358.392,A -85,B 0,C 180,E1 -6225.729,E2 -6225.729} C_VEL
LIN {X 0,Y 496.302,Z 344.378,A -85,B 0,C 180,E1 -6226.042,E2 -6226.042} C_VEL
LIN {X 0,Y 496.893,Z 324.439,A -85,B 0,C 180,E1 -6229.198,E2 -6229.198} C_VEL
LIN {X 0,Y 497.53,Z 305.737,A -85,B 0,C 180,E1 -6232.2,E2 -6232.2} C_VEL
LIN {X 0,Y 497.925,Z 295.005,A -85,B 0,C 180,E1 -6233.947,E2 -6233.947} C_VEL
LIN {X 0,Y 495.837,Z 283.725,A -85,B 0,C 180,E1 -6235.951,E2 -6235.951} C_VEL
LIN {X 0,Y 495.767,Z 283.728,A -85,B 0,C 180,E1 -6238.814,E2 -6238.814} C_VEL
LIN {X 0,Y 495.753,Z 283.732,A -85,B 0,C 180,E1 -6241.724,E2 -6241.724} C_VEL
LIN {X 0,Y 495.764,Z 283.727,A -85,B 0,C 180,E1 -6244.693,E2 -6244.693} C_VEL
LIN {X 0,Y 495.717,Z 283.736,A -85,B 0,C 180,E1 -6247.561,E2 -6247.561} C_VEL
LIN {X 0,Y 495.753,Z 283.733,A -85,B 0,C 180,E1 -6250.046,E2 -6250.046} C_VEL
LIN {X 0,Y 495.711,Z 283.734,A -85,B 0,C 180,E1 -6252.883,E2 -6252.883} C_VEL
LIN {X 0,Y 495.718,Z 283.736,A -85,B 0,C 180,E1 -6255.997,E2 -6255.997} C_VEL
LIN {X 0,Y 495.716,Z 283.733,A -85,B 0,C 180,E1 -6258.711,E2 -6258.711} C_VEL
LIN {X 0,Y 495.739,Z 283.735,A -85,B 0,C 180,E1 -6261.407,E2 -6261.407} C_VEL
LIN {X 0,Y 495.74,Z 283.73,A -85,B 0,C 180,E1 -6264.461,E2 -6264.461} C_VEL
LIN {X 0,Y 495.758,Z 283.735,A -85,B 0,C 180,E1 -6267.405,E2 -6267.405} C_VEL
LIN {X 0,Y 495.749,Z 283.729,A -85,B 0,C 180,E1 -6270.252,E2 -6270.252} C_VEL
LIN {X 0,Y 495.73,Z 283.738,A -85,B 0,C 180,E1 -6273.27,E2 -6273.27} C_VEL
LIN {X 0,Y 495.729,Z 283.734,A -85,B 0,C 180,E1 -6276.612,E2 -6276.612} C_VEL
LIN {X 0,Y 495.77,Z 283.731,A -85,B 0,C 180,E1 -6279.324,E2 -6279.324} C_VEL
LIN {X 0,Y 495.77,Z 283.727,A -85,B 0,C 180,E1 -6281.828,E2 -6281.828} C_VEL
LIN {X 0,Y 495.814,Z 283.724,A -85,B 0,C 180,E1 -6284.549,E2 -6284.549} C_VEL
LIN {X 0,Y 495.819,Z 283.722,A -85,B 0,C 180,E1 -6287.965,E2 -6287.965} C_VEL
LIN {X 0,Y 495.818,Z 283.726,A -85,B 0,C 180,E1 -6291.03,E2 -6291.03} C_VEL
LIN {X 0,Y 495.794,Z 283.725,A -85,B 0,C 180,E1 -6293.489,E2 -6293.489} C_VEL
LIN {X 0,Y 495.703,Z 283.737,A -85,B 0,C 180,E1 -6295.935,E2 -6295.935} C_VEL
LIN {X 0,Y 495.968,Z 283.703,A -85,B 0,C 180,E1 -6297.564,E2 -6297.564} C_VEL
LIN {X 0,Y 495.931,Z 283.711,A -85,B 0,C 180,E1 -6300.812,E2 -6300.812} C_VEL
LIN {X 0,Y 495.962,Z 283.707,A -85,B 0,C 180,E1 -6302.436,E2 -6302.436} C_VEL
LIN {X 0,Y 495.843,Z 283.72,A -85,B 0,C 180,E1 -6305.694,E2 -6305.694} C_VEL
LIN {X 0,Y 495.803,Z 283.726,A -85,B 0,C 180,E1 -6308.149,E2 -6308.149} C_VEL
LIN {X 0,Y 495.84,Z 283.72,A -85,B 0,C 180,E1 -6311.446,E2 -6311.446} C_VEL
LIN {X 0,Y 495.772,Z 283.728,A -85,B 0,C 180,E1 -6314.784,E2 -6314.784} C_VEL
LIN {X 0,Y 495.745,Z 283.732,A -85,B 0,C 180,E1 -6317.32,E2 -6317.32} C_VEL
LIN {X 0,Y 495.758,Z 283.732,A -85,B 0,C 180,E1 -6319.891,E2 -6319.891} C_VEL
LIN {X 0,Y 495.75,Z 283.73,A -85,B 0,C 180,E1 -6322.861,E2 -6322.861} C_VEL
LIN {X 0,Y 495.749,Z 283.734,A -85,B 0,C 180,E1 -6326.07,E2 -6326.07} C_VEL
LIN {X 0,Y 495.735,Z 283.732,A -85,B 0,C 180,E1 -6328.817,E2 -6328.817} C_VEL
LIN {X 0,Y 495.747,Z 283.734,A -85,B 0,C 180,E1 -6331.726,E2 -6331.726} C_VEL
LIN {X 0,Y 495.761,Z 283.729,A -85,B 0,C 180,E1 -6334.694,E2 -6334.694} C_VEL
LIN {X 0,Y 495.715,Z 283.738,A -85,B 0,C 180,E1 -6337.563,E2 -6337.563} C_VEL
LIN {X 0,Y 495.752,Z 283.731,A -85,B 0,C 180,E1 -6340.048,E2 -6340.048} C_VEL
LIN {X 0,Y 495.711,Z 283.738,A -85,B 0,C 180,E1 -6342.885,E2 -6342.885} C_VEL
LIN {X 0,Y 495.723,Z 283.734,A -85,B 0,C 180,E1 -6345.999,E2 -6345.999} C_VEL
LIN {X 0,Y 495.762,Z 283.732,A -85,B 0,C 180,E1 -6349.301,E2 -6349.301} C_VEL
LIN {X 0,Y 495.725,Z 283.734,A -85,B 0,C 180,E1 -6352.439,E2 -6352.439} C_VEL
LIN {X 0,Y 495.768,Z 283.731,A -85,B 0,C 180,E1 -6355.457,E2 -6355.457} C_VEL
LIN {X 0,Y 495.752,Z 283.732,A -85,B 0,C 180,E1 -6358.365,E2 -6358.365} C_VEL
LIN {X 0,Y 495.749,Z 283.73,A -85,B 0,C 180,E1 -6360.752,E2 -6360.752} C_VEL
LIN {X 0,Y 495.092,Z 283.815,A -85,B 0,C 180,E1 -6361.431,E2 -6361.431} C_VEL
LIN {X 0,Y 492.236,Z 284.172,A -85,B 0,C 180,E1 -6362.534,E2 -6362.534} C_VEL
LIN {X 0,Y 489.827,Z 284.47,A -85,B 0,C 180,E1 -6363.422,E2 -6363.422} C_VEL
LIN {X 0,Y 488.808,Z 284.596,A -85,B 0,C 180,E1 -6364.109,E2 -6364.109} C_VEL
LIN {X 0,Y 488.733,Z 284.607,A -85,B 0,C 180,E1 -6364.341,E2 -6364.341} C_VEL
LIN {X 0,Y 488.721,Z 284.608,A -85,B 0,C 180,E1 -6367.154,E2 -6367.154} C_VEL
LIN {X 0,Y 488.728,Z 284.605,A -85,B 0,C 180,E1 -6369.812,E2 -6369.812} C_VEL
LIN {X 0,Y 488.792,Z 284.6,A -85,B 0,C 180,E1 -6371.618,E2 -6371.618} C_VEL
LIN {X 0,Y 488.589,Z 284.77,A -85,B 0,C 180,E1 -6372.743,E2 -6372.743} C_VEL
LIN {X 0,Y 488.88,Z 294.961,A -85,B 0,C 180,E1 -6373.704,E2 -6373.704} C_VEL
LIN {X 0,Y 491.835,Z 314.665,A -85,B 0,C 180,E1 -6374.101,E2 -6374.101} C_VEL
LIN {X 0,Y 491.182,Z 408.282,A -85,B 0,C 180,E1 -6375.5,E2 -6375.5} C_VEL
LIN {X 0,Y 490.965,Z 421.546,A -85,B 0,C 180,E1 -6375.864,E2 -6375.864} C_VEL
LIN {X 0,Y 490.628,Z 434.016,A -85,B 0,C 180,E1 -6376.382,E2 -6376.382} C_VEL
LIN {X 0,Y 490.328,Z 445.305,A -85,B 0,C 180,E1 -6377.012,E2 -6377.012} C_VEL
LIN {X 0,Y 489.988,Z 456.217,A -85,B 0,C 180,E1 -6377.787,E2 -6377.787} C_VEL
LIN {X 0,Y 489.554,Z 466.674,A -85,B 0,C 180,E1 -6378.721,E2 -6378.721} C_VEL
LIN {X 0,Y 489.183,Z 475.236,A -85,B 0,C 180,E1 -6379.655,E2 -6379.655} C_VEL
LIN {X 0,Y 488.827,Z 484.541,A -85,B 0,C 180,E1 -6380.901,E2 -6380.901} C_VEL
LIN {X 0,Y 488.491,Z 491.946,A -85,B 0,C 180,E1 -6382.145,E2 -6382.145} C_VEL
LIN {X 0,Y 488.31,Z 497.891,A -85,B 0,C 180,E1 -6383.389,E2 -6383.389} C_VEL
LIN {X 0,Y 488.08,Z 502.597,A -85,B 0,C 180,E1 -6384.63,E2 -6384.63} C_VEL
LIN {X 0,Y 488.114,Z 506.188,A -85,B 0,C 180,E1 -6385.872,E2 -6385.872} C_VEL
LIN {X 0,Y 488.055,Z 508.041,A -85,B 0,C 180,E1 -6386.699,E2 -6386.699} C_VEL
LIN {X 0,Y 488.006,Z 509.461,A -85,B 0,C 180,E1 -6387.525,E2 -6387.525} C_VEL
LIN {X 0,Y 487.84,Z 511.074,A -85,B 0,C 180,E1 -6389.175,E2 -6389.175} C_VEL
LIN {X 0,Y 487.829,Z 511.311,A -85,B 0,C 180,E1 -6390.001,E2 -6390.001} C_VEL
LIN {X 0,Y 487.894,Z 510.542,A -85,B 0,C 180,E1 -6391.652,E2 -6391.652} C_VEL
LIN {X 0,Y 488.007,Z 509.579,A -85,B 0,C 180,E1 -6392.477,E2 -6392.477} C_VEL
LIN {X 0,Y 488.056,Z 508.224,A -85,B 0,C 180,E1 -6393.303,E2 -6393.303} C_VEL
LIN {X 0,Y 488.089,Z 505.375,A -85,B 0,C 180,E1 -6394.543,E2 -6394.543} C_VEL
LIN {X 0,Y 488.203,Z 501.499,A -85,B 0,C 180,E1 -6395.784,E2 -6395.784} C_VEL
LIN {X 0,Y 488.33,Z 496.485,A -85,B 0,C 180,E1 -6397.027,E2 -6397.027} C_VEL
LIN {X 0,Y 488.562,Z 490.156,A -85,B 0,C 180,E1 -6398.272,E2 -6398.272} C_VEL
LIN {X 0,Y 488.874,Z 482.283,A -85,B 0,C 180,E1 -6399.517,E2 -6399.517} C_VEL
LIN {X 0,Y 489.22,Z 474.236,A -85,B 0,C 180,E1 -6400.555,E2 -6400.555} C_VEL
LIN {X 0,Y 489.62,Z 464.37,A -85,B 0,C 180,E1 -6401.594,E2 -6401.594} C_VEL
LIN {X 0,Y 490.056,Z 453.158,A -85,B 0,C 180,E1 -6402.538,E2 -6402.538} C_VEL
LIN {X 0,Y 490.396,Z 442.442,A -85,B 0,C 180,E1 -6403.257,E2 -6403.257} C_VEL
LIN {X 0,Y 490.731,Z 430.309,A -85,B 0,C 180,E1 -6403.881,E2 -6403.881} C_VEL
LIN {X 0,Y 491.065,Z 416.933,A -85,B 0,C 180,E1 -6404.373,E2 -6404.373} C_VEL
LIN {X 0,Y 491.238,Z 403.283,A -85,B 0,C 180,E1 -6404.685,E2 -6404.685} C_VEL
LIN {X 0,Y 491.752,Z 313.181,A -85,B 0,C 180,E1 -6406.014,E2 -6406.014} C_VEL
LIN {X 0,Y 488.849,Z 294.733,A -85,B 0,C 180,E1 -6406.409,E2 -6406.409} C_VEL
LIN {X 0,Y 488.566,Z 284.633,A -85,B 0,C 180,E1 -6407.368,E2 -6407.368} C_VEL
LIN {X 0,Y 488.774,Z 284.602,A -85,B 0,C 180,E1 -6408.442,E2 -6408.442} C_VEL
LIN {X 0,Y 488.712,Z 284.61,A -85,B 0,C 180,E1 -6411.071,E2 -6411.071} C_VEL
LIN {X 0,Y 488.684,Z 284.614,A -85,B 0,C 180,E1 -6413.747,E2 -6413.747} C_VEL
LIN {X 0,Y 488.796,Z 284.598,A -85,B 0,C 180,E1 -6416.944,E2 -6416.944} C_VEL
LIN {X 0,Y 488.713,Z 284.606,A -85,B 0,C 180,E1 -6420.363,E2 -6420.363} C_VEL
LIN {X 0,Y 488.734,Z 284.609,A -85,B 0,C 180,E1 -6423.484,E2 -6423.484} C_VEL
LIN {X 0,Y 488.687,Z 284.609,A -85,B 0,C 180,E1 -6426.355,E2 -6426.355} C_VEL
LIN {X 0,Y 488.706,Z 284.613,A -85,B 0,C 180,E1 -6429.255,E2 -6429.255} C_VEL
LIN {X 0,Y 488.712,Z 284.608,A -85,B 0,C 180,E1 -6431.6,E2 -6431.6} C_VEL
LIN {X 0,Y 488.717,Z 284.608,A -85,B 0,C 180,E1 -6434.802,E2 -6434.802} C_VEL
